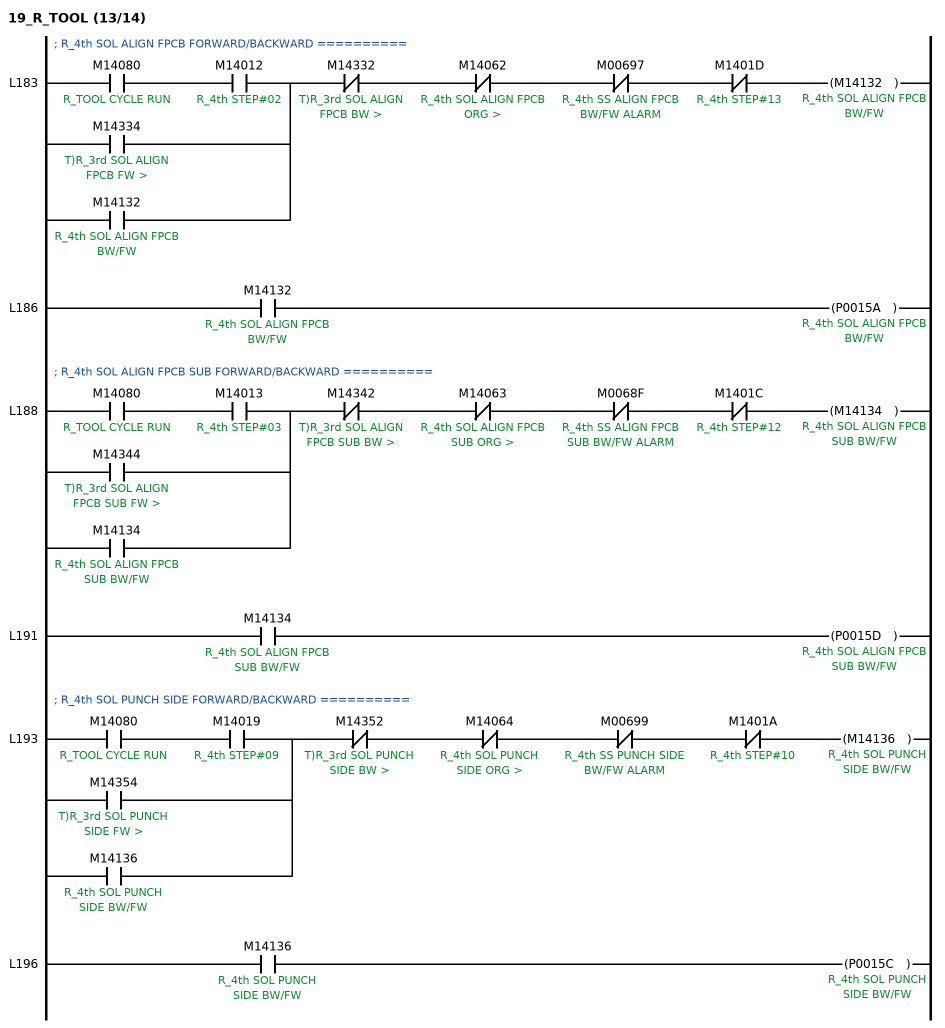
[picture p192: 19_R_TOOL rungs L183-L196]
// R_4th SOL ALIGN FPCB FORWARD/BACKWARD ==========
; L183
LOAD      M14080	// R_TOOL CYCLE RUN
AND       M14012	// R_4th STEP#02
OR        M14334	// T)R_3rd SOL ALIGN FPCB FW >
OR        M14132	// R_4th SOL ALIGN FPCB BW/FW
AND NOT   M14332	// T)R_3rd SOL ALIGN FPCB BW >
AND NOT   M14062	// R_4th SOL ALIGN FPCB ORG >
AND NOT   M00697	// R_4th SS ALIGN FPCB BW/FW ALARM
AND NOT   M1401D	// R_4th STEP#13
OUT       M14132	// R_4th SOL ALIGN FPCB BW/FW
; L186
LOAD      M14132	// R_4th SOL ALIGN FPCB BW/FW
OUT       P0015A	// R_4th SOL ALIGN FPCB BW/FW
// R_4th SOL ALIGN FPCB SUB FORWARD/BACKWARD ==========
; L188
LOAD      M14080	// R_TOOL CYCLE RUN
AND       M14013	// R_4th STEP#03
OR        M14344	// T)R_3rd SOL ALIGN FPCB SUB FW >
OR        M14134	// R_4th SOL ALIGN FPCB SUB BW/FW
AND NOT   M14342	// T)R_3rd SOL ALIGN FPCB SUB BW >
AND NOT   M14063	// R_4th SOL ALIGN FPCB SUB ORG >
AND NOT   M0068F	// R_4th SS ALIGN FPCB SUB BW/FW ALARM
AND NOT   M1401C	// R_4th STEP#12
OUT       M14134	// R_4th SOL ALIGN FPCB SUB BW/FW
; L191
LOAD      M14134	// R_4th SOL ALIGN FPCB SUB BW/FW
OUT       P0015D	// R_4th SOL ALIGN FPCB SUB BW/FW
// R_4th SOL PUNCH SIDE FORWARD/BACKWARD ==========
; L193
LOAD      M14080	// R_TOOL CYCLE RUN
AND       M14019	// R_4th STEP#09
OR        M14354	// T)R_3rd SOL PUNCH SIDE FW >
OR        M14136	// R_4th SOL PUNCH SIDE BW/FW
AND NOT   M14352	// T)R_3rd SOL PUNCH SIDE BW >
AND NOT   M14064	// R_4th SOL PUNCH SIDE ORG >
AND NOT   M00699	// R_4th SS PUNCH SIDE BW/FW ALARM
AND NOT   M1401A	// R_4th STEP#10
OUT       M14136	// R_4th SOL PUNCH SIDE BW/FW
; L196
LOAD      M14136	// R_4th SOL PUNCH SIDE BW/FW
OUT       P0015C	// R_4th SOL PUNCH SIDE BW/FW

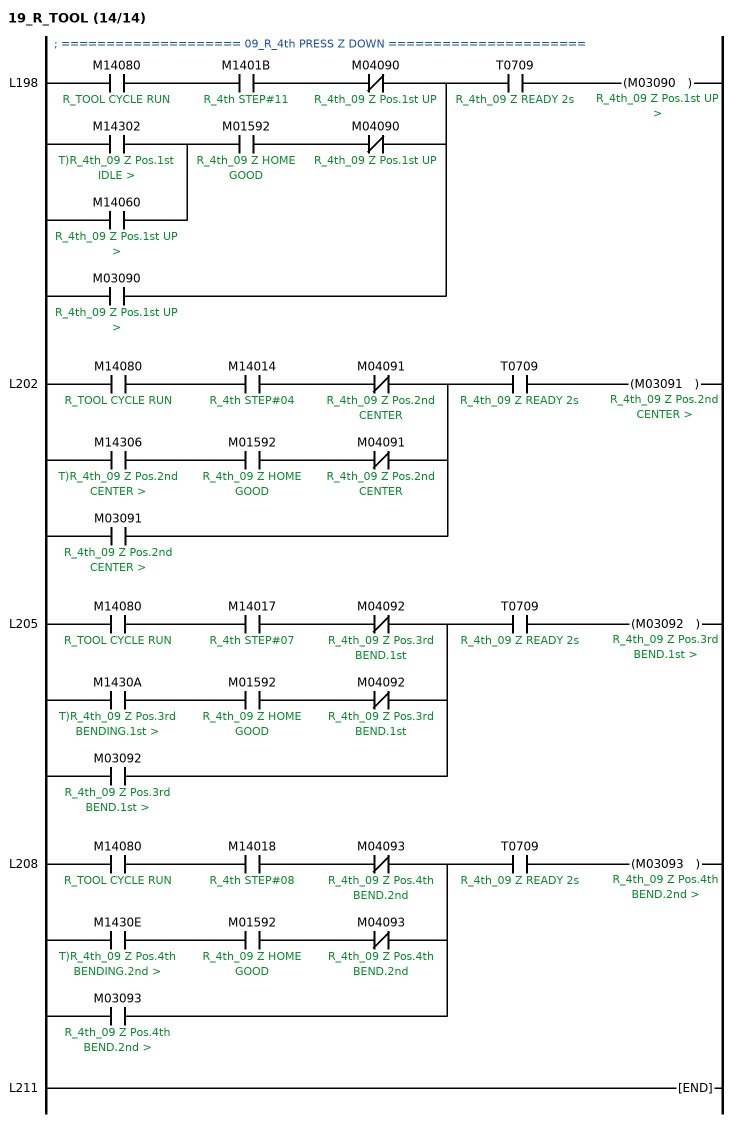
// ==================== 09_R_4th PRESS Z DOWN ======================
; L198
LOAD      M14080	// R_TOOL CYCLE RUN
AND       M1401B	// R_4th STEP#11
AND NOT   M04090	// R_4th_09 Z Pos.1st UP
LOAD      M14302	// T)R_4th_09 Z Pos.1st IDLE >
OR        M14060	// R_4th_09 Z Pos.1st UP >
AND       M01592	// R_4th_09 Z HOME GOOD
AND NOT   M04090	// R_4th_09 Z Pos.1st UP
OR LOAD
OR        M03090	// R_4th_09 Z Pos.1st UP >
AND       T0709	// R_4th_09 Z READY 2s
OUT       M03090	// R_4th_09 Z Pos.1st UP >
; L202
LOAD      M14080	// R_TOOL CYCLE RUN
AND       M14014	// R_4th STEP#04
AND NOT   M04091	// R_4th_09 Z Pos.2nd CENTER
LOAD      M14306	// T)R_4th_09 Z Pos.2nd CENTER >
AND       M01592	// R_4th_09 Z HOME GOOD
AND NOT   M04091	// R_4th_09 Z Pos.2nd CENTER
OR LOAD
OR        M03091	// R_4th_09 Z Pos.2nd CENTER >
AND       T0709	// R_4th_09 Z READY 2s
OUT       M03091	// R_4th_09 Z Pos.2nd CENTER >
; L205
LOAD      M14080	// R_TOOL CYCLE RUN
AND       M14017	// R_4th STEP#07
AND NOT   M04092	// R_4th_09 Z Pos.3rd BEND.1st
LOAD      M1430A	// T)R_4th_09 Z Pos.3rd BENDING.1st >
AND       M01592	// R_4th_09 Z HOME GOOD
AND NOT   M04092	// R_4th_09 Z Pos.3rd BEND.1st
OR LOAD
OR        M03092	// R_4th_09 Z Pos.3rd BEND.1st >
AND       T0709	// R_4th_09 Z READY 2s
OUT       M03092	// R_4th_09 Z Pos.3rd BEND.1st >
; L208
LOAD      M14080	// R_TOOL CYCLE RUN
AND       M14018	// R_4th STEP#08
AND NOT   M04093	// R_4th_09 Z Pos.4th BEND.2nd
LOAD      M1430E	// T)R_4th_09 Z Pos.4th BENDING.2nd >
AND       M01592	// R_4th_09 Z HOME GOOD
AND NOT   M04093	// R_4th_09 Z Pos.4th BEND.2nd
OR LOAD
OR        M03093	// R_4th_09 Z Pos.4th BEND.2nd >
AND       T0709	// R_4th_09 Z READY 2s
OUT       M03093	// R_4th_09 Z Pos.4th BEND.2nd >
; L211
END

PROGRAM 20_R_PP (task: ½ºÄµ ÇÁ·Î±×·¥)

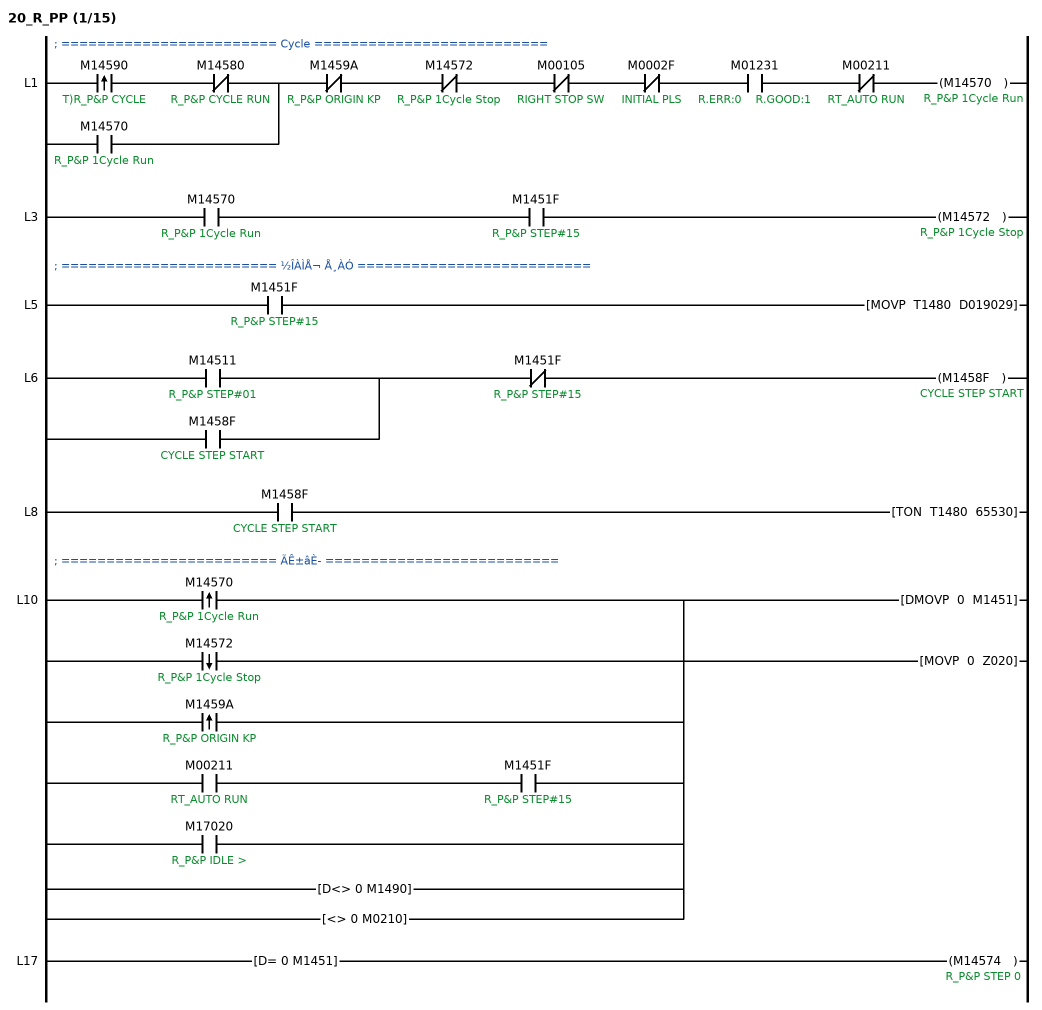
// ======================== Cycle ==========================
; L1
LOADP     M14590	// T)R_P&P CYCLE
AND NOT   M14580	// R_P&P CYCLE RUN
OR        M14570	// R_P&P 1Cycle Run
AND NOT   M1459A	// R_P&P ORIGIN KP
AND NOT   M14572	// R_P&P 1Cycle Stop
AND NOT   M00105	// RIGHT STOP SW
AND NOT   M0002F	// INITIAL PLS
AND       M01231	// R.ERR:0    R.GOOD:1
AND NOT   M00211	// RT_AUTO RUN
OUT       M14570	// R_P&P 1Cycle Run
; L3
LOAD      M14570	// R_P&P 1Cycle Run
AND       M1451F	// R_P&P STEP#15
OUT       M14572	// R_P&P 1Cycle Stop
// ======================== ½ÎÀÌÅ¬ Å¸ÀÓ ==========================
; L5
LOAD      M1451F	// R_P&P STEP#15
MOVP      T1480 D019029
; L6
LOAD      M14511	// R_P&P STEP#01
OR        M1458F	// CYCLE STEP START
AND NOT   M1451F	// R_P&P STEP#15
OUT       M1458F	// CYCLE STEP START
; L8
LOAD      M1458F	// CYCLE STEP START
TON       T1480 65530
// ======================== ÃÊ±âÈ­ ==========================
; L10
LOADP     M14570	// R_P&P 1Cycle Run
ORN       M14572	// R_P&P 1Cycle Stop
ORP       M1459A	// R_P&P ORIGIN KP
LOAD      M00211	// RT_AUTO RUN
AND       M1451F	// R_P&P STEP#15
OR LOAD
OR        M17020	// R_P&P IDLE >
ORD<>     0 M1490
OR<>      0 M0210
DMOVP     0 M1451
MOVP      0 Z020
; L17
LOADD=    0 M1451
OUT       M14574	// R_P&P STEP 0

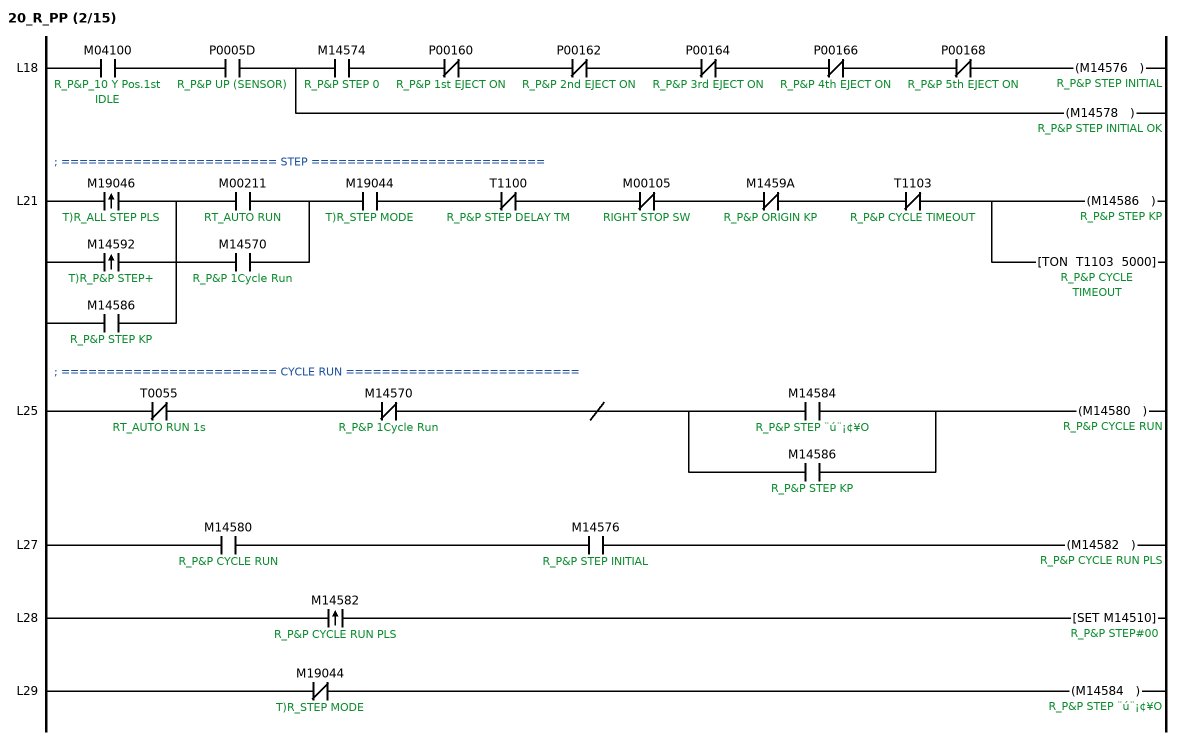
; L18
LOAD      M04100	// R_P&P_10 Y Pos.1st IDLE
AND       P0005D	// R_P&P UP (SENSOR)
MPUSH
AND       M14574	// R_P&P STEP 0
AND NOT   P00160	// R_P&P 1st EJECT ON
AND NOT   P00162	// R_P&P 2nd EJECT ON
AND NOT   P00164	// R_P&P 3rd EJECT ON
AND NOT   P00166	// R_P&P 4th EJECT ON
AND NOT   P00168	// R_P&P 5th EJECT ON
OUT       M14576	// R_P&P STEP INITIAL
MPOP
OUT       M14578	// R_P&P STEP INITIAL OK
// ======================== STEP ==========================
; L21
LOADP     M19046	// T)R_ALL STEP PLS
ORP       M14592	// T)R_P&P STEP+
OR        M14586	// R_P&P STEP KP
LOAD      M00211	// RT_AUTO RUN
OR        M14570	// R_P&P 1Cycle Run
AND LOAD
AND       M19044	// T)R_STEP MODE
AND NOT   T1100	// R_P&P STEP DELAY TM
AND NOT   M00105	// RIGHT STOP SW
AND NOT   M1459A	// R_P&P ORIGIN KP
AND NOT   T1103	// R_P&P CYCLE TIMEOUT
OUT       M14586	// R_P&P STEP KP
TON       T1103 5000	// R_P&P CYCLE TIMEOUT
// ======================== CYCLE RUN ==========================
; L25
LOAD NOT  T0055	// RT_AUTO RUN 1s
AND NOT   M14570	// R_P&P 1Cycle Run
NOT
LOAD      M14584	// R_P&P STEP ¨ú¨¡¢¥O
OR        M14586	// R_P&P STEP KP
AND LOAD
OUT       M14580	// R_P&P CYCLE RUN
; L27
LOAD      M14580	// R_P&P CYCLE RUN
AND       M14576	// R_P&P STEP INITIAL
OUT       M14582	// R_P&P CYCLE RUN PLS
; L28
LOADP     M14582	// R_P&P CYCLE RUN PLS
SET       M14510	// R_P&P STEP#00
; L29
LOAD NOT  M19044	// T)R_STEP MODE
OUT       M14584	// R_P&P STEP ¨ú¨¡¢¥O

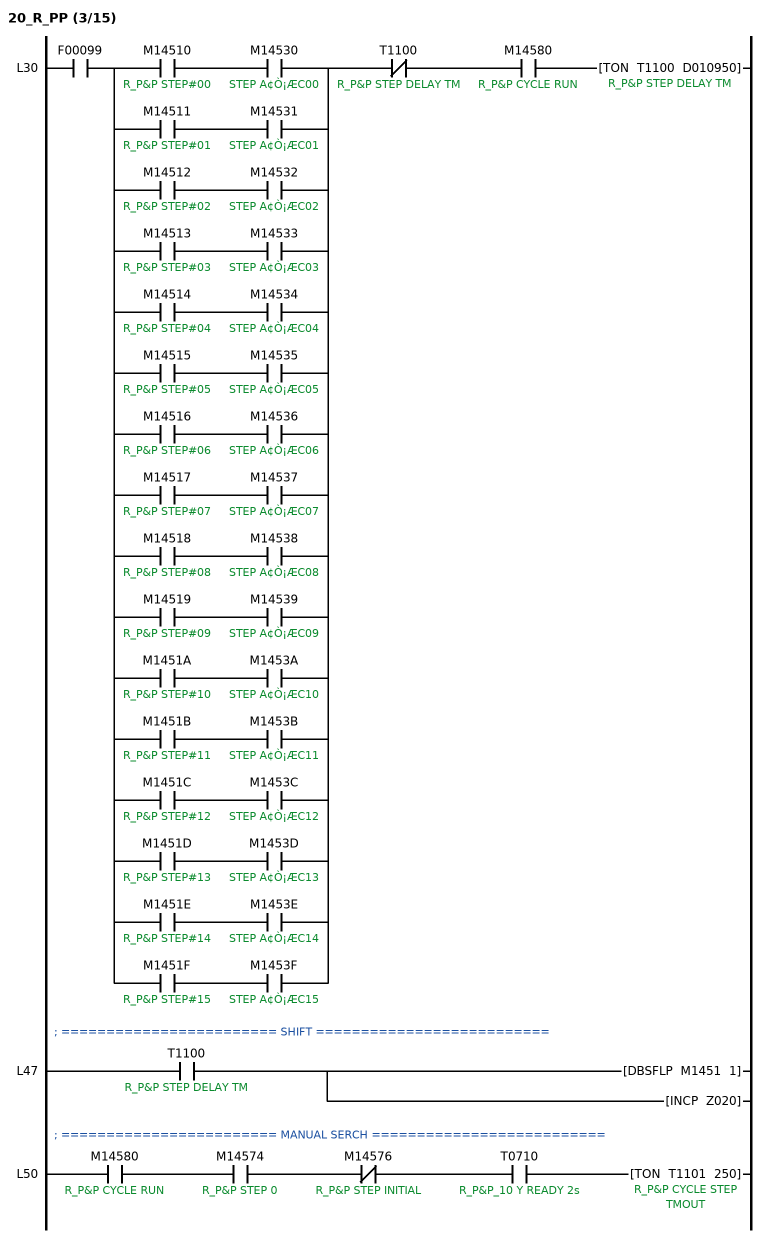
; L30
LOAD      F00099
LOAD      M14510	// R_P&P STEP#00
AND       M14530	// STEP A¢Ò¡ÆC00
LOAD      M14511	// R_P&P STEP#01
AND       M14531	// STEP A¢Ò¡ÆC01
OR LOAD
LOAD      M14512	// R_P&P STEP#02
AND       M14532	// STEP A¢Ò¡ÆC02
OR LOAD
LOAD      M14513	// R_P&P STEP#03
AND       M14533	// STEP A¢Ò¡ÆC03
OR LOAD
LOAD      M14514	// R_P&P STEP#04
AND       M14534	// STEP A¢Ò¡ÆC04
OR LOAD
LOAD      M14515	// R_P&P STEP#05
AND       M14535	// STEP A¢Ò¡ÆC05
OR LOAD
LOAD      M14516	// R_P&P STEP#06
AND       M14536	// STEP A¢Ò¡ÆC06
OR LOAD
LOAD      M14517	// R_P&P STEP#07
AND       M14537	// STEP A¢Ò¡ÆC07
OR LOAD
LOAD      M14518	// R_P&P STEP#08
AND       M14538	// STEP A¢Ò¡ÆC08
OR LOAD
LOAD      M14519	// R_P&P STEP#09
AND       M14539	// STEP A¢Ò¡ÆC09
OR LOAD
LOAD      M1451A	// R_P&P STEP#10
AND       M1453A	// STEP A¢Ò¡ÆC10
OR LOAD
LOAD      M1451B	// R_P&P STEP#11
AND       M1453B	// STEP A¢Ò¡ÆC11
OR LOAD
LOAD      M1451C	// R_P&P STEP#12
AND       M1453C	// STEP A¢Ò¡ÆC12
OR LOAD
LOAD      M1451D	// R_P&P STEP#13
AND       M1453D	// STEP A¢Ò¡ÆC13
OR LOAD
LOAD      M1451E	// R_P&P STEP#14
AND       M1453E	// STEP A¢Ò¡ÆC14
OR LOAD
LOAD      M1451F	// R_P&P STEP#15
AND       M1453F	// STEP A¢Ò¡ÆC15
OR LOAD
AND LOAD
AND NOT   T1100	// R_P&P STEP DELAY TM
AND       M14580	// R_P&P CYCLE RUN
TON       T1100 D010950	// R_P&P STEP DELAY TM
// ======================== SHIFT ==========================
; L47
LOAD      T1100	// R_P&P STEP DELAY TM
DBSFLP    M1451 1
INCP      Z020
// ======================== MANUAL SERCH ==========================
; L50
LOAD      M14580	// R_P&P CYCLE RUN
AND       M14574	// R_P&P STEP 0
AND NOT   M14576	// R_P&P STEP INITIAL
AND       T0710	// R_P&P_10 Y READY 2s
TON       T1101 250	// R_P&P CYCLE STEP TMOUT

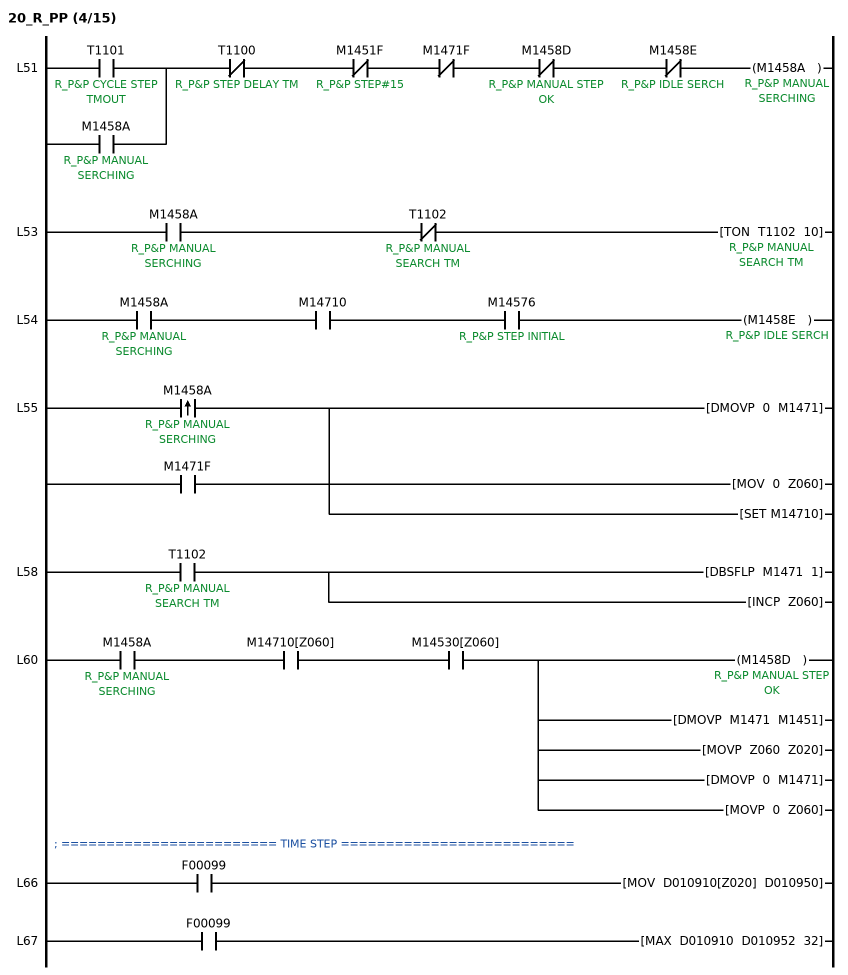
; L51
LOAD      T1101	// R_P&P CYCLE STEP TMOUT
OR        M1458A	// R_P&P MANUAL SERCHING
AND NOT   T1100	// R_P&P STEP DELAY TM
AND NOT   M1451F	// R_P&P STEP#15
AND NOT   M1471F
AND NOT   M1458D	// R_P&P MANUAL STEP OK
AND NOT   M1458E	// R_P&P IDLE SERCH
OUT       M1458A	// R_P&P MANUAL SERCHING
; L53
LOAD      M1458A	// R_P&P MANUAL SERCHING
AND NOT   T1102	// R_P&P MANUAL SEARCH TM
TON       T1102 10	// R_P&P MANUAL SEARCH TM
; L54
LOAD      M1458A	// R_P&P MANUAL SERCHING
AND       M14710
AND       M14576	// R_P&P STEP INITIAL
OUT       M1458E	// R_P&P IDLE SERCH
; L55
LOADP     M1458A	// R_P&P MANUAL SERCHING
OR        M1471F
DMOVP     0 M1471
MOV       0 Z060
SET       M14710
; L58
LOAD      T1102	// R_P&P MANUAL SEARCH TM
DBSFLP    M1471 1
INCP      Z060
; L60
LOAD      M1458A	// R_P&P MANUAL SERCHING
AND       M14710[Z060]
AND       M14530[Z060]
OUT       M1458D	// R_P&P MANUAL STEP OK
DMOVP     M1471 M1451
MOVP      Z060 Z020
DMOVP     0 M1471
MOVP      0 Z060
// ======================== TIME STEP ==========================
; L66
LOAD      F00099
MOV       D010910[Z020] D010950
; L67
LOAD      F00099
MAX       D010910 D010952 32

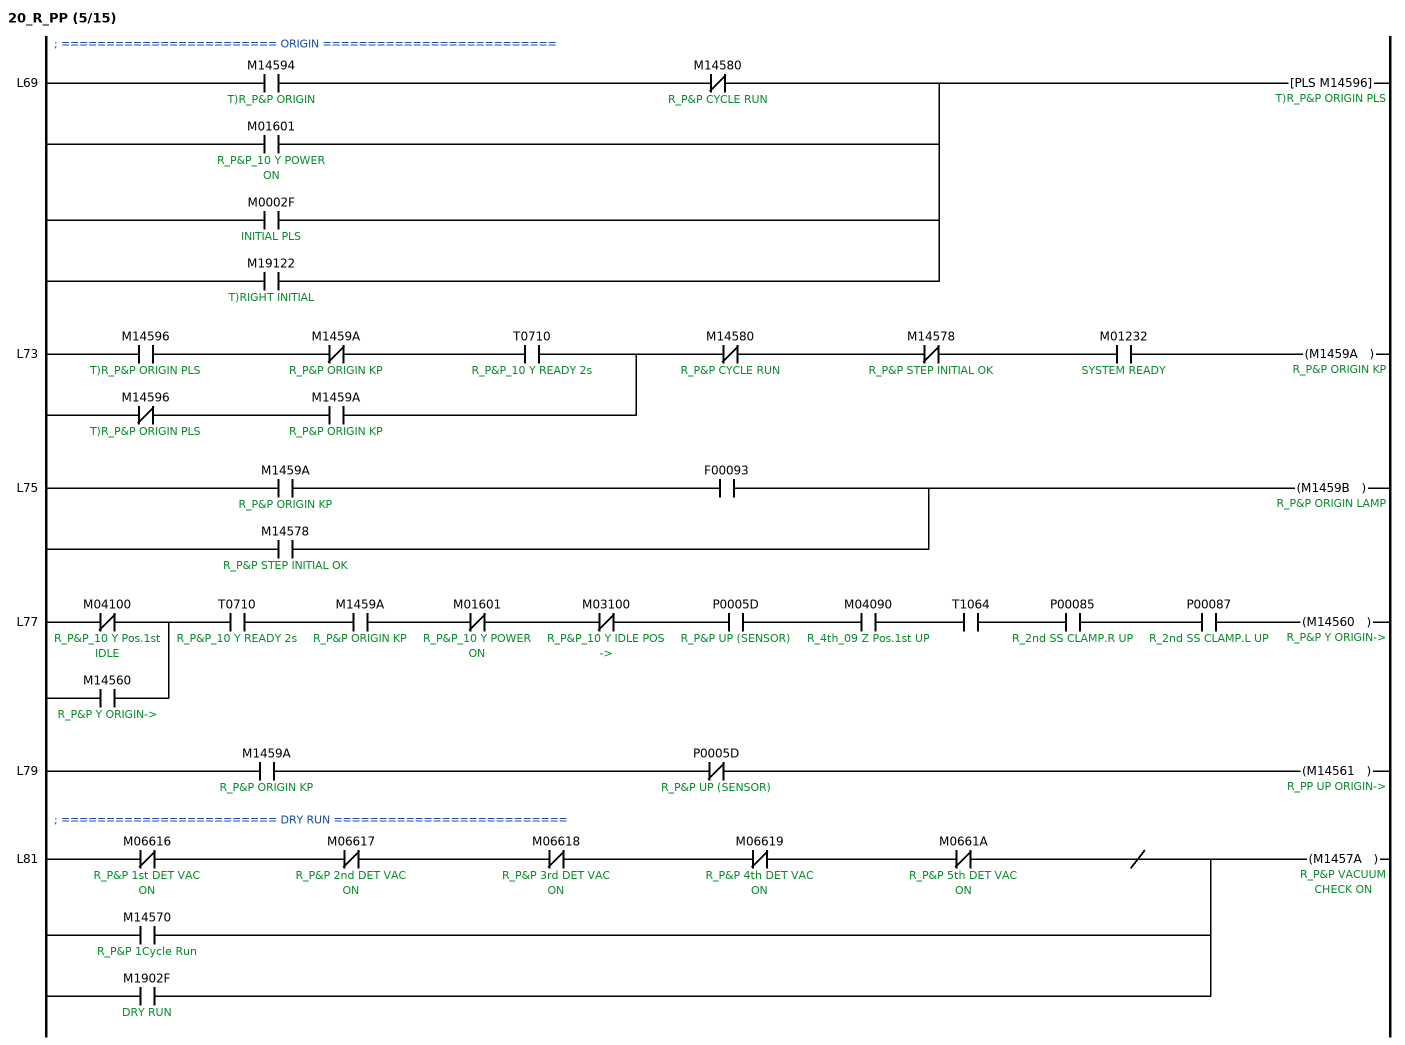
// ======================== ORIGIN ==========================
; L69
LOAD      M14594	// T)R_P&P ORIGIN
AND NOT   M14580	// R_P&P CYCLE RUN
OR        M01601	// R_P&P_10 Y POWER ON
OR        M0002F	// INITIAL PLS
OR        M19122	// T)RIGHT INITIAL
OUTP      M14596	// T)R_P&P ORIGIN PLS
; L73
LOAD      M14596	// T)R_P&P ORIGIN PLS
AND NOT   M1459A	// R_P&P ORIGIN KP
AND       T0710	// R_P&P_10 Y READY 2s
LOAD NOT  M14596	// T)R_P&P ORIGIN PLS
AND       M1459A	// R_P&P ORIGIN KP
OR LOAD
AND NOT   M14580	// R_P&P CYCLE RUN
AND NOT   M14578	// R_P&P STEP INITIAL OK
AND       M01232	// SYSTEM READY
OUT       M1459A	// R_P&P ORIGIN KP
; L75
LOAD      M1459A	// R_P&P ORIGIN KP
AND       F00093
OR        M14578	// R_P&P STEP INITIAL OK
OUT       M1459B	// R_P&P ORIGIN LAMP
; L77
LOAD NOT  M04100	// R_P&P_10 Y Pos.1st IDLE
OR        M14560	// R_P&P Y ORIGIN->
AND       T0710	// R_P&P_10 Y READY 2s
AND       M1459A	// R_P&P ORIGIN KP
AND NOT   M01601	// R_P&P_10 Y POWER ON
AND NOT   M03100	// R_P&P_10 Y IDLE POS ->
AND       P0005D	// R_P&P UP (SENSOR)
AND       M04090	// R_4th_09 Z Pos.1st UP
AND       T1064
AND       P00085	// R_2nd SS CLAMP.R UP
AND       P00087	// R_2nd SS CLAMP.L UP
OUT       M14560	// R_P&P Y ORIGIN->
; L79
LOAD      M1459A	// R_P&P ORIGIN KP
AND NOT   P0005D	// R_P&P UP (SENSOR)
OUT       M14561	// R_PP UP ORIGIN->
// ======================== DRY RUN ==========================
; L81
LOAD NOT  M06616	// R_P&P 1st DET VAC ON
AND NOT   M06617	// R_P&P 2nd DET VAC ON
AND NOT   M06618	// R_P&P 3rd DET VAC ON
AND NOT   M06619	// R_P&P 4th DET VAC ON
AND NOT   M0661A	// R_P&P 5th DET VAC ON
NOT
OR        M14570	// R_P&P 1Cycle Run
OR        M1902F	// DRY RUN
OUT       M1457A	// R_P&P VACUUM CHECK ON

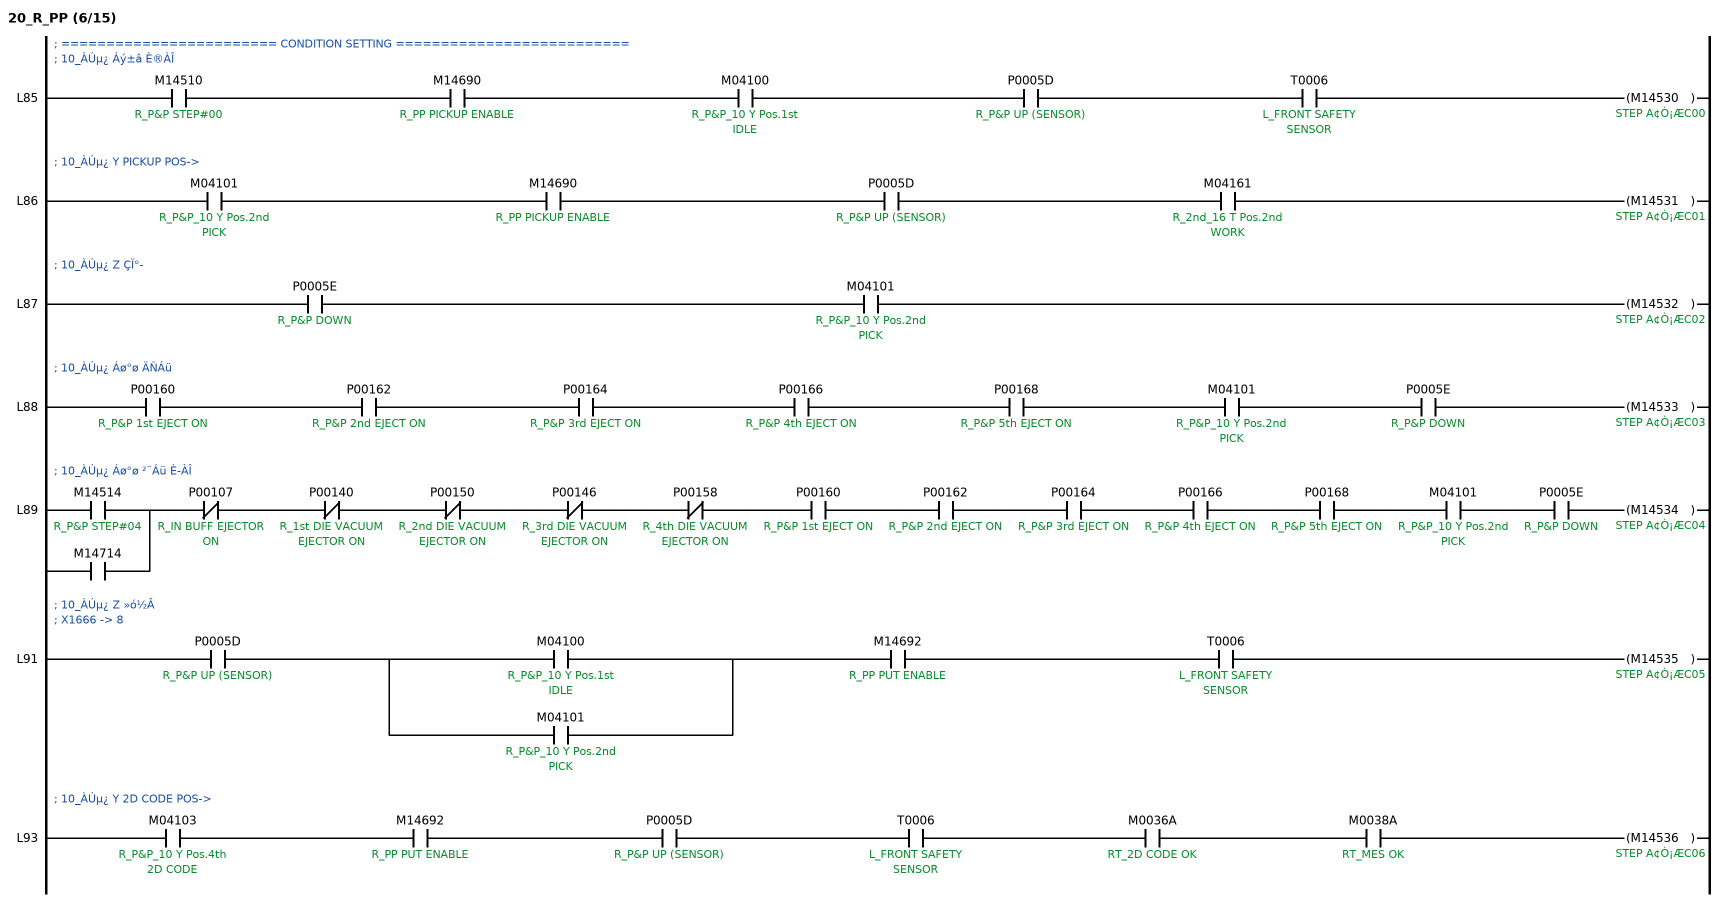
// ======================== CONDITION SETTING ==========================
; L85
LOAD      M14510	// R_P&P STEP#00
AND       M14690	// R_PP PICKUP ENABLE
AND       M04100	// R_P&P_10 Y Pos.1st IDLE
AND       P0005D	// R_P&P UP (SENSOR)
AND       T0006	// L_FRONT SAFETY SENSOR
OUT       M14530	// STEP A¢Ò¡ÆC00
// output comment: 10_ÀÚµ¿ Áý±â È®ÀÎ
; L86
LOAD      M04101	// R_P&P_10 Y Pos.2nd PICK
AND       M14690	// R_PP PICKUP ENABLE
AND       P0005D	// R_P&P UP (SENSOR)
AND       M04161	// R_2nd_16 T Pos.2nd WORK
OUT       M14531	// STEP A¢Ò¡ÆC01
// output comment: 10_ÀÚµ¿ Y PICKUP POS->
; L87
LOAD      P0005E	// R_P&P DOWN
AND       M04101	// R_P&P_10 Y Pos.2nd PICK
OUT       M14532	// STEP A¢Ò¡ÆC02
// output comment: 10_ÀÚµ¿ Z ÇÏ°­
; L88
LOAD      P00160	// R_P&P 1st EJECT ON
AND       P00162	// R_P&P 2nd EJECT ON
AND       P00164	// R_P&P 3rd EJECT ON
AND       P00166	// R_P&P 4th EJECT ON
AND       P00168	// R_P&P 5th EJECT ON
AND       M04101	// R_P&P_10 Y Pos.2nd PICK
AND       P0005E	// R_P&P DOWN
OUT       M14533	// STEP A¢Ò¡ÆC03
// output comment: 10_ÀÚµ¿ Áø°ø ÄÑÁü
; L89
LOAD      M14514	// R_P&P STEP#04
OR        M14714
AND NOT   P00107	// R_IN BUFF EJECTOR ON
AND NOT   P00140	// R_1st DIE VACUUM EJECTOR ON
AND NOT   P00150	// R_2nd DIE VACUUM EJECTOR ON
AND NOT   P00146	// R_3rd DIE VACUUM EJECTOR ON
AND NOT   P00158	// R_4th DIE VACUUM EJECTOR ON
AND       P00160	// R_P&P 1st EJECT ON
AND       P00162	// R_P&P 2nd EJECT ON
AND       P00164	// R_P&P 3rd EJECT ON
AND       P00166	// R_P&P 4th EJECT ON
AND       P00168	// R_P&P 5th EJECT ON
AND       M04101	// R_P&P_10 Y Pos.2nd PICK
AND       P0005E	// R_P&P DOWN
OUT       M14534	// STEP A¢Ò¡ÆC04
// output comment: 10_ÀÚµ¿ Áø°ø ²¨Áü È­ÀÎ
; L91
LOAD      P0005D	// R_P&P UP (SENSOR)
LOAD      M04100	// R_P&P_10 Y Pos.1st IDLE
OR        M04101	// R_P&P_10 Y Pos.2nd PICK
AND LOAD
AND       M14692	// R_PP PUT ENABLE
AND       T0006	// L_FRONT SAFETY SENSOR
OUT       M14535	// STEP A¢Ò¡ÆC05
// output comment: 10_ÀÚµ¿ Z »ó½Â X1666 -> 8
; L93
LOAD      M04103	// R_P&P_10 Y Pos.4th 2D CODE
AND       M14692	// R_PP PUT ENABLE
AND       P0005D	// R_P&P UP (SENSOR)
AND       T0006	// L_FRONT SAFETY SENSOR
AND       M0036A	// RT_2D CODE OK
AND       M0038A	// RT_MES OK
OUT       M14536	// STEP A¢Ò¡ÆC06
// output comment: 10_ÀÚµ¿ Y 2D CODE POS->

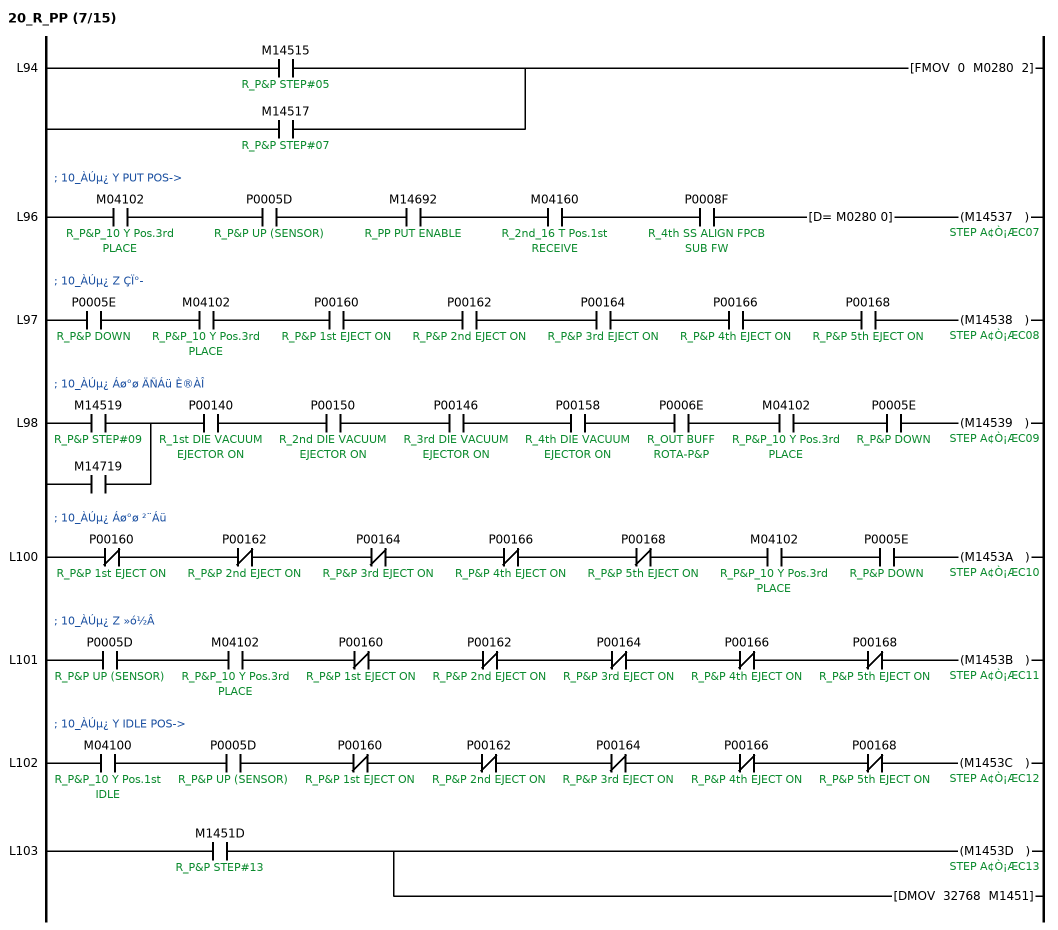
; L94
LOAD      M14515	// R_P&P STEP#05
OR        M14517	// R_P&P STEP#07
FMOV      0 M0280 2
; L96
LOAD      M04102	// R_P&P_10 Y Pos.3rd PLACE
AND       P0005D	// R_P&P UP (SENSOR)
AND       M14692	// R_PP PUT ENABLE
AND       M04160	// R_2nd_16 T Pos.1st RECEIVE
AND       P0008F	// R_4th SS ALIGN FPCB SUB FW
ANDD=     M0280 0
OUT       M14537	// STEP A¢Ò¡ÆC07
// output comment: 10_ÀÚµ¿ Y PUT POS->
; L97
LOAD      P0005E	// R_P&P DOWN
AND       M04102	// R_P&P_10 Y Pos.3rd PLACE
AND       P00160	// R_P&P 1st EJECT ON
AND       P00162	// R_P&P 2nd EJECT ON
AND       P00164	// R_P&P 3rd EJECT ON
AND       P00166	// R_P&P 4th EJECT ON
AND       P00168	// R_P&P 5th EJECT ON
OUT       M14538	// STEP A¢Ò¡ÆC08
// output comment: 10_ÀÚµ¿ Z ÇÏ°­
; L98
LOAD      M14519	// R_P&P STEP#09
OR        M14719
AND       P00140	// R_1st DIE VACUUM EJECTOR ON
AND       P00150	// R_2nd DIE VACUUM EJECTOR ON
AND       P00146	// R_3rd DIE VACUUM EJECTOR ON
AND       P00158	// R_4th DIE VACUUM EJECTOR ON
AND       P0006E	// R_OUT BUFF ROTA-P&P
AND       M04102	// R_P&P_10 Y Pos.3rd PLACE
AND       P0005E	// R_P&P DOWN
OUT       M14539	// STEP A¢Ò¡ÆC09
// output comment: 10_ÀÚµ¿ Áø°ø ÄÑÁü È®ÀÎ
; L100
LOAD NOT  P00160	// R_P&P 1st EJECT ON
AND NOT   P00162	// R_P&P 2nd EJECT ON
AND NOT   P00164	// R_P&P 3rd EJECT ON
AND NOT   P00166	// R_P&P 4th EJECT ON
AND NOT   P00168	// R_P&P 5th EJECT ON
AND       M04102	// R_P&P_10 Y Pos.3rd PLACE
AND       P0005E	// R_P&P DOWN
OUT       M1453A	// STEP A¢Ò¡ÆC10
// output comment: 10_ÀÚµ¿ Áø°ø ²¨Áü
; L101
LOAD      P0005D	// R_P&P UP (SENSOR)
AND       M04102	// R_P&P_10 Y Pos.3rd PLACE
AND NOT   P00160	// R_P&P 1st EJECT ON
AND NOT   P00162	// R_P&P 2nd EJECT ON
AND NOT   P00164	// R_P&P 3rd EJECT ON
AND NOT   P00166	// R_P&P 4th EJECT ON
AND NOT   P00168	// R_P&P 5th EJECT ON
OUT       M1453B	// STEP A¢Ò¡ÆC11
// output comment: 10_ÀÚµ¿ Z »ó½Â
; L102
LOAD      M04100	// R_P&P_10 Y Pos.1st IDLE
AND       P0005D	// R_P&P UP (SENSOR)
AND NOT   P00160	// R_P&P 1st EJECT ON
AND NOT   P00162	// R_P&P 2nd EJECT ON
AND NOT   P00164	// R_P&P 3rd EJECT ON
AND NOT   P00166	// R_P&P 4th EJECT ON
AND NOT   P00168	// R_P&P 5th EJECT ON
OUT       M1453C	// STEP A¢Ò¡ÆC12
// output comment: 10_ÀÚµ¿ Y IDLE POS->
; L103
LOAD      M1451D	// R_P&P STEP#13
OUT       M1453D	// STEP A¢Ò¡ÆC13
DMOV      32768 M1451

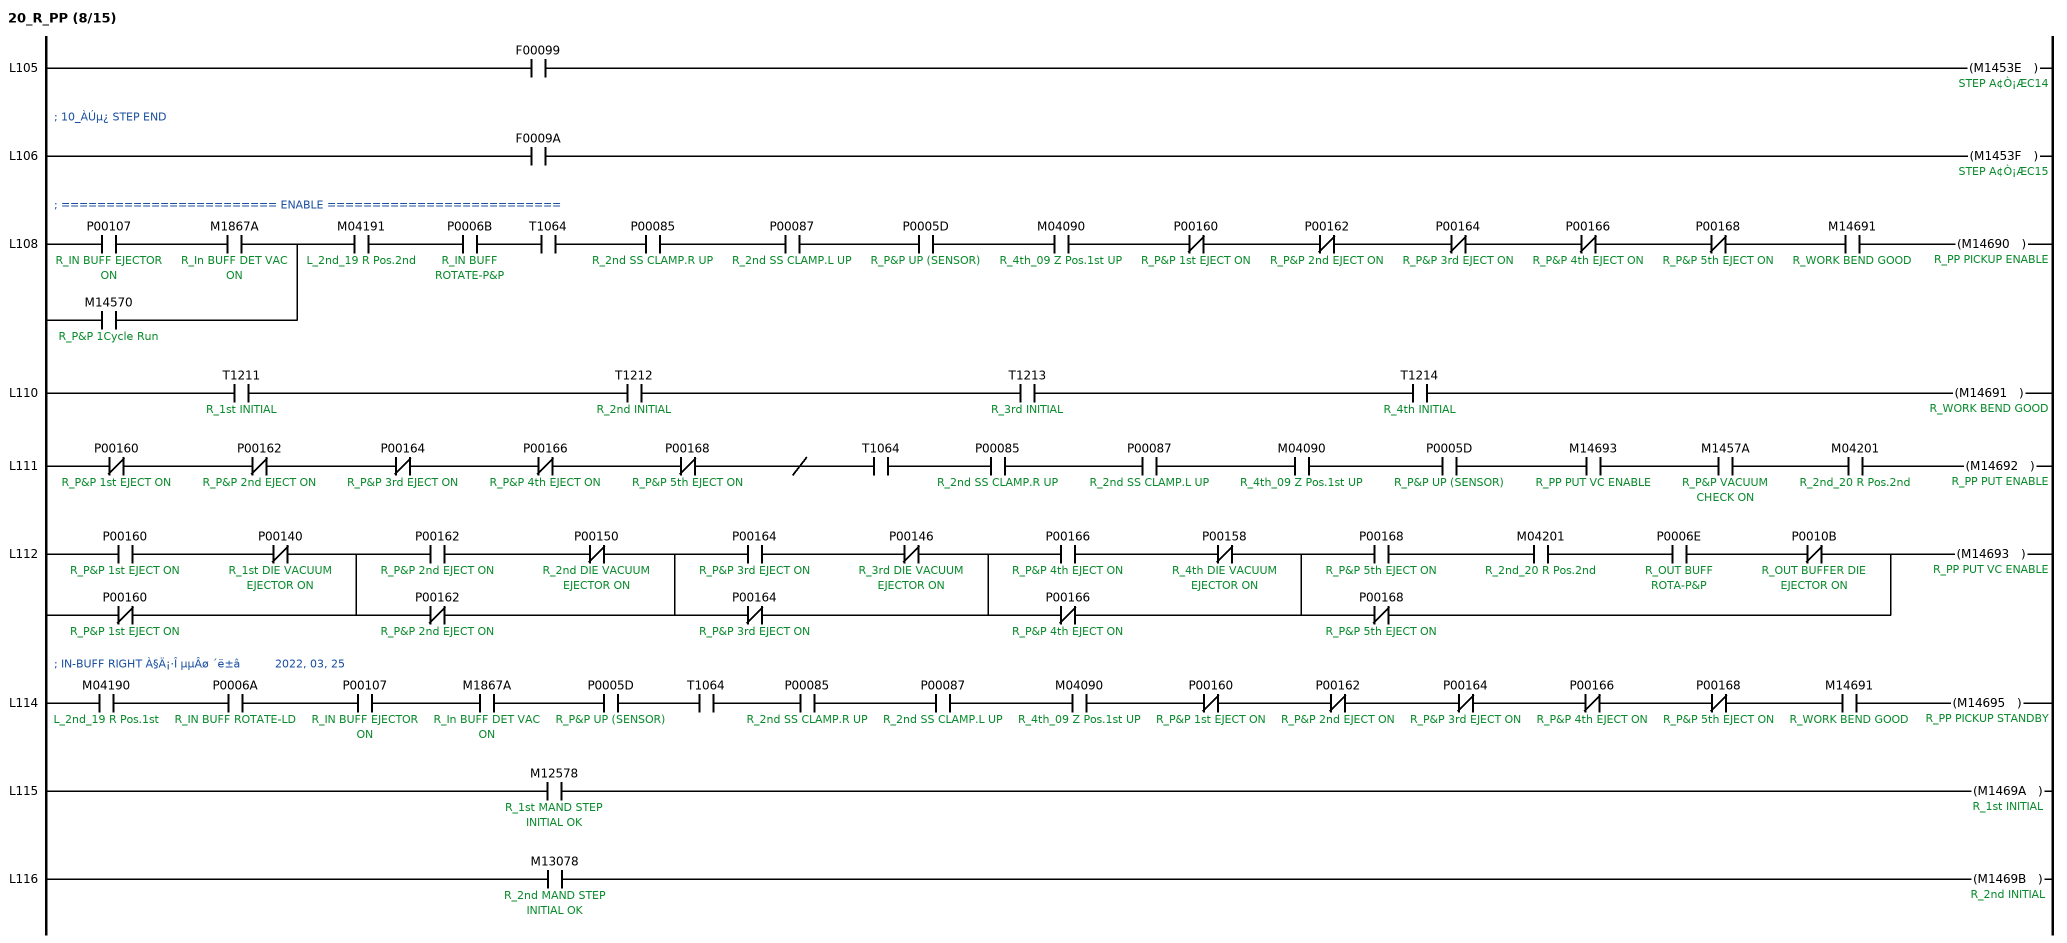
; L105
LOAD      F00099
OUT       M1453E	// STEP A¢Ò¡ÆC14
; L106
LOAD      F0009A
OUT       M1453F	// STEP A¢Ò¡ÆC15
// output comment: 10_ÀÚµ¿ STEP END
// ======================== ENABLE ==========================
; L108
LOAD      P00107	// R_IN BUFF EJECTOR ON
AND       M1867A	// R_In BUFF DET VAC ON
OR        M14570	// R_P&P 1Cycle Run
AND       M04191	// L_2nd_19 R Pos.2nd
AND       P0006B	// R_IN BUFF ROTATE-P&P
AND       T1064
AND       P00085	// R_2nd SS CLAMP.R UP
AND       P00087	// R_2nd SS CLAMP.L UP
AND       P0005D	// R_P&P UP (SENSOR)
AND       M04090	// R_4th_09 Z Pos.1st UP
AND NOT   P00160	// R_P&P 1st EJECT ON
AND NOT   P00162	// R_P&P 2nd EJECT ON
AND NOT   P00164	// R_P&P 3rd EJECT ON
AND NOT   P00166	// R_P&P 4th EJECT ON
AND NOT   P00168	// R_P&P 5th EJECT ON
AND       M14691	// R_WORK BEND GOOD
OUT       M14690	// R_PP PICKUP ENABLE
; L110
LOAD      T1211	// R_1st INITIAL
AND       T1212	// R_2nd INITIAL
AND       T1213	// R_3rd INITIAL
AND       T1214	// R_4th INITIAL
OUT       M14691	// R_WORK BEND GOOD
; L111
LOAD NOT  P00160	// R_P&P 1st EJECT ON
AND NOT   P00162	// R_P&P 2nd EJECT ON
AND NOT   P00164	// R_P&P 3rd EJECT ON
AND NOT   P00166	// R_P&P 4th EJECT ON
AND NOT   P00168	// R_P&P 5th EJECT ON
NOT
AND       T1064
AND       P00085	// R_2nd SS CLAMP.R UP
AND       P00087	// R_2nd SS CLAMP.L UP
AND       M04090	// R_4th_09 Z Pos.1st UP
AND       P0005D	// R_P&P UP (SENSOR)
AND       M14693	// R_PP PUT VC ENABLE
AND       M1457A	// R_P&P VACUUM CHECK ON
AND       M04201	// R_2nd_20 R Pos.2nd
OUT       M14692	// R_PP PUT ENABLE
; L112
LOAD      P00160	// R_P&P 1st EJECT ON
AND NOT   P00140	// R_1st DIE VACUUM EJECTOR ON
OR NOT    P00160	// R_P&P 1st EJECT ON
LOAD      P00162	// R_P&P 2nd EJECT ON
AND NOT   P00150	// R_2nd DIE VACUUM EJECTOR ON
OR NOT    P00162	// R_P&P 2nd EJECT ON
AND LOAD
LOAD      P00164	// R_P&P 3rd EJECT ON
AND NOT   P00146	// R_3rd DIE VACUUM EJECTOR ON
OR NOT    P00164	// R_P&P 3rd EJECT ON
AND LOAD
LOAD      P00166	// R_P&P 4th EJECT ON
AND NOT   P00158	// R_4th DIE VACUUM EJECTOR ON
OR NOT    P00166	// R_P&P 4th EJECT ON
AND LOAD
LOAD      P00168	// R_P&P 5th EJECT ON
AND       M04201	// R_2nd_20 R Pos.2nd
AND       P0006E	// R_OUT BUFF ROTA-P&P
AND NOT   P0010B	// R_OUT BUFFER DIE EJECTOR ON
OR NOT    P00168	// R_P&P 5th EJECT ON
AND LOAD
OUT       M14693	// R_PP PUT VC ENABLE
; L114
LOAD      M04190	// L_2nd_19 R Pos.1st 
AND       P0006A	// R_IN BUFF ROTATE-LD
AND       P00107	// R_IN BUFF EJECTOR ON
AND       M1867A	// R_In BUFF DET VAC ON
AND       P0005D	// R_P&P UP (SENSOR)
AND       T1064
AND       P00085	// R_2nd SS CLAMP.R UP
AND       P00087	// R_2nd SS CLAMP.L UP
AND       M04090	// R_4th_09 Z Pos.1st UP
AND NOT   P00160	// R_P&P 1st EJECT ON
AND NOT   P00162	// R_P&P 2nd EJECT ON
AND NOT   P00164	// R_P&P 3rd EJECT ON
AND NOT   P00166	// R_P&P 4th EJECT ON
AND NOT   P00168	// R_P&P 5th EJECT ON
AND       M14691	// R_WORK BEND GOOD
OUT       M14695	// R_PP PICKUP STANDBY
// output comment: IN-BUFF RIGHT À§Ä¡·Î µµÂø ´ë±â          2022, 03, 25
; L115
LOAD      M12578	// R_1st MAND STEP INITIAL OK
OUT       M1469A	// R_1st INITIAL
; L116
LOAD      M13078	// R_2nd MAND STEP INITIAL OK
OUT       M1469B	// R_2nd INITIAL

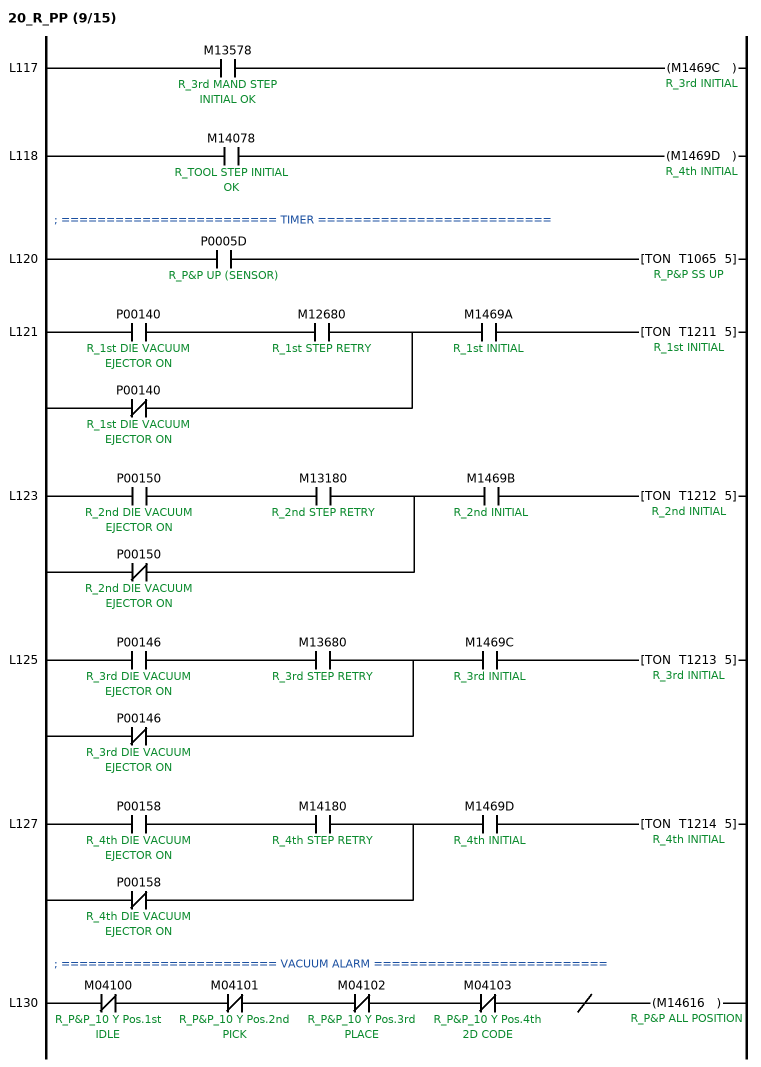
; L117
LOAD      M13578	// R_3rd MAND STEP INITIAL OK
OUT       M1469C	// R_3rd INITIAL
; L118
LOAD      M14078	// R_TOOL STEP INITIAL OK
OUT       M1469D	// R_4th INITIAL
// ======================== TIMER ==========================
; L120
LOAD      P0005D	// R_P&P UP (SENSOR)
TON       T1065 5	// R_P&P SS UP
; L121
LOAD      P00140	// R_1st DIE VACUUM EJECTOR ON
AND       M12680	// R_1st STEP RETRY
OR NOT    P00140	// R_1st DIE VACUUM EJECTOR ON
AND       M1469A	// R_1st INITIAL
TON       T1211 5	// R_1st INITIAL
; L123
LOAD      P00150	// R_2nd DIE VACUUM EJECTOR ON
AND       M13180	// R_2nd STEP RETRY
OR NOT    P00150	// R_2nd DIE VACUUM EJECTOR ON
AND       M1469B	// R_2nd INITIAL
TON       T1212 5	// R_2nd INITIAL
; L125
LOAD      P00146	// R_3rd DIE VACUUM EJECTOR ON
AND       M13680	// R_3rd STEP RETRY
OR NOT    P00146	// R_3rd DIE VACUUM EJECTOR ON
AND       M1469C	// R_3rd INITIAL
TON       T1213 5	// R_3rd INITIAL
; L127
LOAD      P00158	// R_4th DIE VACUUM EJECTOR ON
AND       M14180	// R_4th STEP RETRY
OR NOT    P00158	// R_4th DIE VACUUM EJECTOR ON
AND       M1469D	// R_4th INITIAL
TON       T1214 5	// R_4th INITIAL
// ======================== VACUUM ALARM ==========================
; L130
LOAD NOT  M04100	// R_P&P_10 Y Pos.1st IDLE
AND NOT   M04101	// R_P&P_10 Y Pos.2nd PICK
AND NOT   M04102	// R_P&P_10 Y Pos.3rd PLACE
AND NOT   M04103	// R_P&P_10 Y Pos.4th 2D CODE
NOT
OUT       M14616	// R_P&P ALL POSITION

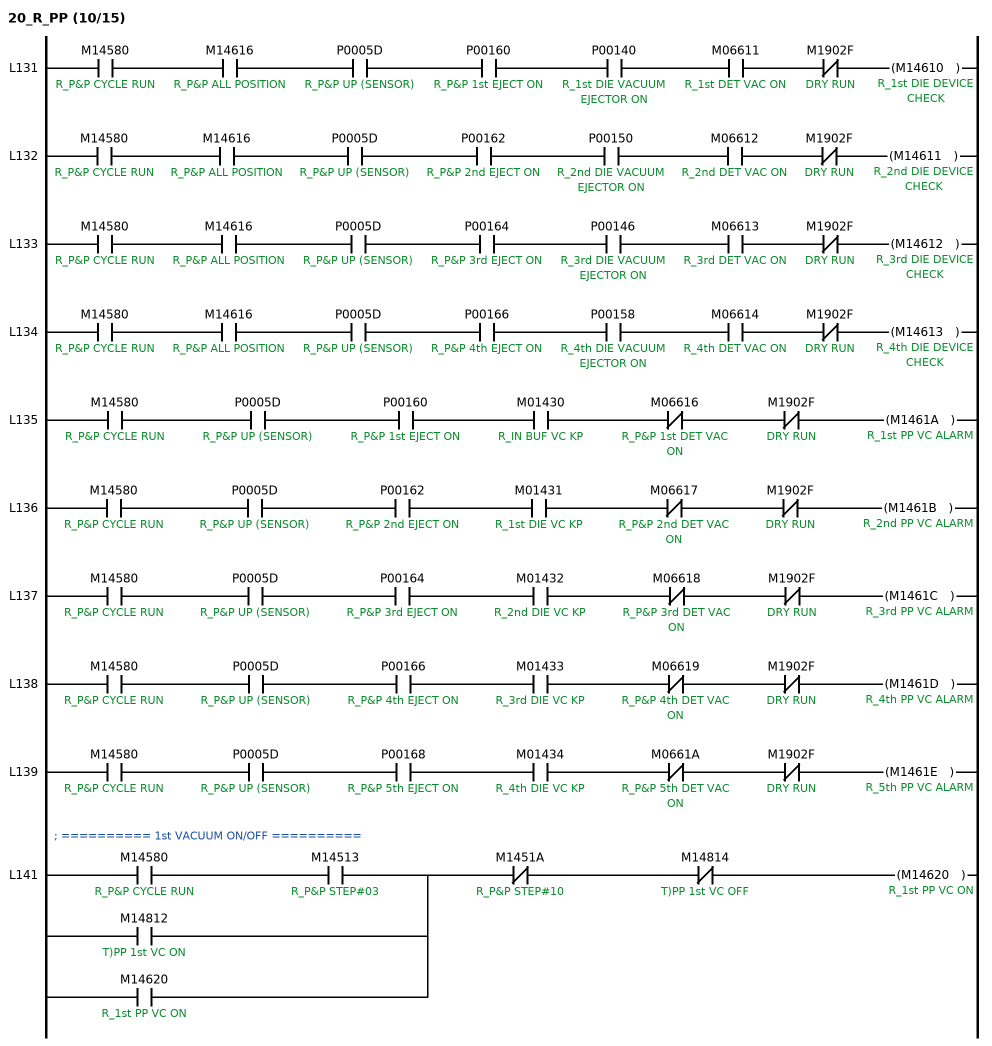
; L131
LOAD      M14580	// R_P&P CYCLE RUN
AND       M14616	// R_P&P ALL POSITION
AND       P0005D	// R_P&P UP (SENSOR)
AND       P00160	// R_P&P 1st EJECT ON
AND       P00140	// R_1st DIE VACUUM EJECTOR ON
AND       M06611	// R_1st DET VAC ON
AND NOT   M1902F	// DRY RUN
OUT       M14610	// R_1st DIE DEVICE CHECK
; L132
LOAD      M14580	// R_P&P CYCLE RUN
AND       M14616	// R_P&P ALL POSITION
AND       P0005D	// R_P&P UP (SENSOR)
AND       P00162	// R_P&P 2nd EJECT ON
AND       P00150	// R_2nd DIE VACUUM EJECTOR ON
AND       M06612	// R_2nd DET VAC ON
AND NOT   M1902F	// DRY RUN
OUT       M14611	// R_2nd DIE DEVICE CHECK
; L133
LOAD      M14580	// R_P&P CYCLE RUN
AND       M14616	// R_P&P ALL POSITION
AND       P0005D	// R_P&P UP (SENSOR)
AND       P00164	// R_P&P 3rd EJECT ON
AND       P00146	// R_3rd DIE VACUUM EJECTOR ON
AND       M06613	// R_3rd DET VAC ON
AND NOT   M1902F	// DRY RUN
OUT       M14612	// R_3rd DIE DEVICE CHECK
; L134
LOAD      M14580	// R_P&P CYCLE RUN
AND       M14616	// R_P&P ALL POSITION
AND       P0005D	// R_P&P UP (SENSOR)
AND       P00166	// R_P&P 4th EJECT ON
AND       P00158	// R_4th DIE VACUUM EJECTOR ON
AND       M06614	// R_4th DET VAC ON
AND NOT   M1902F	// DRY RUN
OUT       M14613	// R_4th DIE DEVICE CHECK
; L135
LOAD      M14580	// R_P&P CYCLE RUN
AND       P0005D	// R_P&P UP (SENSOR)
AND       P00160	// R_P&P 1st EJECT ON
AND       M01430	// R_IN BUF VC KP
AND NOT   M06616	// R_P&P 1st DET VAC ON
AND NOT   M1902F	// DRY RUN
OUT       M1461A	// R_1st PP VC ALARM
; L136
LOAD      M14580	// R_P&P CYCLE RUN
AND       P0005D	// R_P&P UP (SENSOR)
AND       P00162	// R_P&P 2nd EJECT ON
AND       M01431	// R_1st DIE VC KP
AND NOT   M06617	// R_P&P 2nd DET VAC ON
AND NOT   M1902F	// DRY RUN
OUT       M1461B	// R_2nd PP VC ALARM
; L137
LOAD      M14580	// R_P&P CYCLE RUN
AND       P0005D	// R_P&P UP (SENSOR)
AND       P00164	// R_P&P 3rd EJECT ON
AND       M01432	// R_2nd DIE VC KP
AND NOT   M06618	// R_P&P 3rd DET VAC ON
AND NOT   M1902F	// DRY RUN
OUT       M1461C	// R_3rd PP VC ALARM
; L138
LOAD      M14580	// R_P&P CYCLE RUN
AND       P0005D	// R_P&P UP (SENSOR)
AND       P00166	// R_P&P 4th EJECT ON
AND       M01433	// R_3rd DIE VC KP
AND NOT   M06619	// R_P&P 4th DET VAC ON
AND NOT   M1902F	// DRY RUN
OUT       M1461D	// R_4th PP VC ALARM
; L139
LOAD      M14580	// R_P&P CYCLE RUN
AND       P0005D	// R_P&P UP (SENSOR)
AND       P00168	// R_P&P 5th EJECT ON
AND       M01434	// R_4th DIE VC KP
AND NOT   M0661A	// R_P&P 5th DET VAC ON
AND NOT   M1902F	// DRY RUN
OUT       M1461E	// R_5th PP VC ALARM
// ========== 1st VACUUM ON/OFF ==========
; L141
LOAD      M14580	// R_P&P CYCLE RUN
AND       M14513	// R_P&P STEP#03
OR        M14812	// T)PP 1st VC ON
OR        M14620	// R_1st PP VC ON
AND NOT   M1451A	// R_P&P STEP#10
AND NOT   M14814	// T)PP 1st VC OFF
OUT       M14620	// R_1st PP VC ON

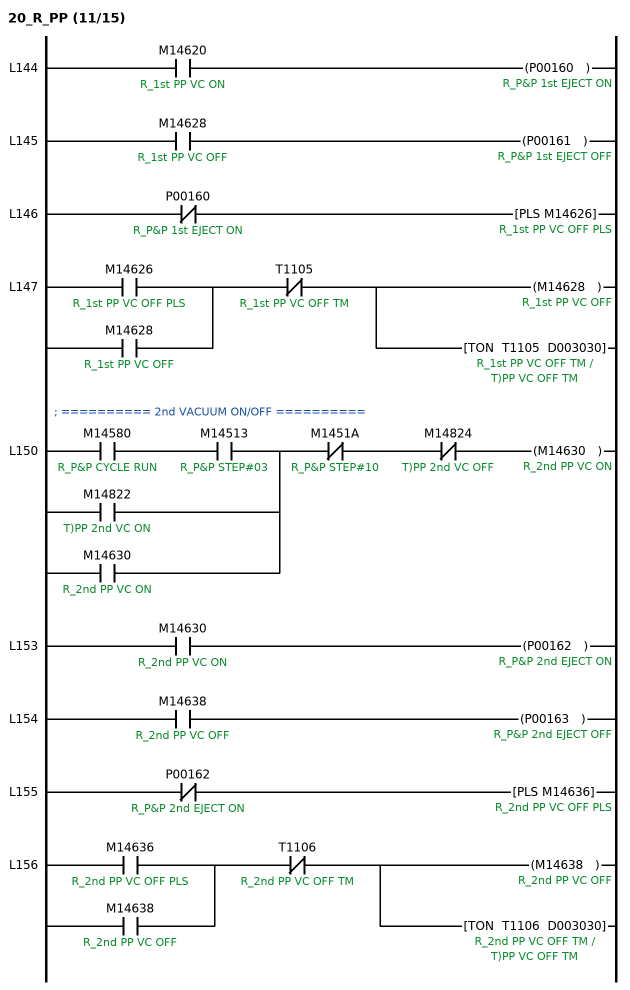
; L144
LOAD      M14620	// R_1st PP VC ON
OUT       P00160	// R_P&P 1st EJECT ON
; L145
LOAD      M14628	// R_1st PP VC OFF
OUT       P00161	// R_P&P 1st EJECT OFF
; L146
LOAD NOT  P00160	// R_P&P 1st EJECT ON
OUTP      M14626	// R_1st PP VC OFF PLS
; L147
LOAD      M14626	// R_1st PP VC OFF PLS
OR        M14628	// R_1st PP VC OFF
AND NOT   T1105	// R_1st PP VC OFF TM
OUT       M14628	// R_1st PP VC OFF
TON       T1105 D003030	// R_1st PP VC OFF TM / T)PP VC OFF TM
// ========== 2nd VACUUM ON/OFF ==========
; L150
LOAD      M14580	// R_P&P CYCLE RUN
AND       M14513	// R_P&P STEP#03
OR        M14822	// T)PP 2nd VC ON
OR        M14630	// R_2nd PP VC ON
AND NOT   M1451A	// R_P&P STEP#10
AND NOT   M14824	// T)PP 2nd VC OFF
OUT       M14630	// R_2nd PP VC ON
; L153
LOAD      M14630	// R_2nd PP VC ON
OUT       P00162	// R_P&P 2nd EJECT ON
; L154
LOAD      M14638	// R_2nd PP VC OFF
OUT       P00163	// R_P&P 2nd EJECT OFF
; L155
LOAD NOT  P00162	// R_P&P 2nd EJECT ON
OUTP      M14636	// R_2nd PP VC OFF PLS
; L156
LOAD      M14636	// R_2nd PP VC OFF PLS
OR        M14638	// R_2nd PP VC OFF
AND NOT   T1106	// R_2nd PP VC OFF TM
OUT       M14638	// R_2nd PP VC OFF
TON       T1106 D003030	// R_2nd PP VC OFF TM / T)PP VC OFF TM

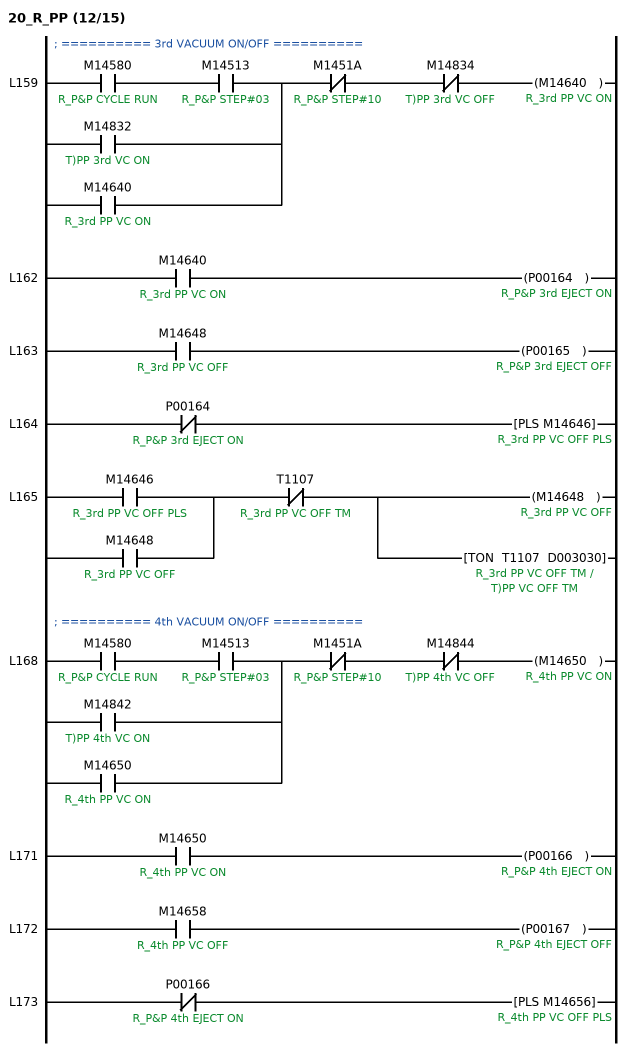
// ========== 3rd VACUUM ON/OFF ==========
; L159
LOAD      M14580	// R_P&P CYCLE RUN
AND       M14513	// R_P&P STEP#03
OR        M14832	// T)PP 3rd VC ON
OR        M14640	// R_3rd PP VC ON
AND NOT   M1451A	// R_P&P STEP#10
AND NOT   M14834	// T)PP 3rd VC OFF
OUT       M14640	// R_3rd PP VC ON
; L162
LOAD      M14640	// R_3rd PP VC ON
OUT       P00164	// R_P&P 3rd EJECT ON
; L163
LOAD      M14648	// R_3rd PP VC OFF
OUT       P00165	// R_P&P 3rd EJECT OFF
; L164
LOAD NOT  P00164	// R_P&P 3rd EJECT ON
OUTP      M14646	// R_3rd PP VC OFF PLS
; L165
LOAD      M14646	// R_3rd PP VC OFF PLS
OR        M14648	// R_3rd PP VC OFF
AND NOT   T1107	// R_3rd PP VC OFF TM
OUT       M14648	// R_3rd PP VC OFF
TON       T1107 D003030	// R_3rd PP VC OFF TM / T)PP VC OFF TM
// ========== 4th VACUUM ON/OFF ==========
; L168
LOAD      M14580	// R_P&P CYCLE RUN
AND       M14513	// R_P&P STEP#03
OR        M14842	// T)PP 4th VC ON
OR        M14650	// R_4th PP VC ON
AND NOT   M1451A	// R_P&P STEP#10
AND NOT   M14844	// T)PP 4th VC OFF
OUT       M14650	// R_4th PP VC ON
; L171
LOAD      M14650	// R_4th PP VC ON
OUT       P00166	// R_P&P 4th EJECT ON
; L172
LOAD      M14658	// R_4th PP VC OFF
OUT       P00167	// R_P&P 4th EJECT OFF
; L173
LOAD NOT  P00166	// R_P&P 4th EJECT ON
OUTP      M14656	// R_4th PP VC OFF PLS

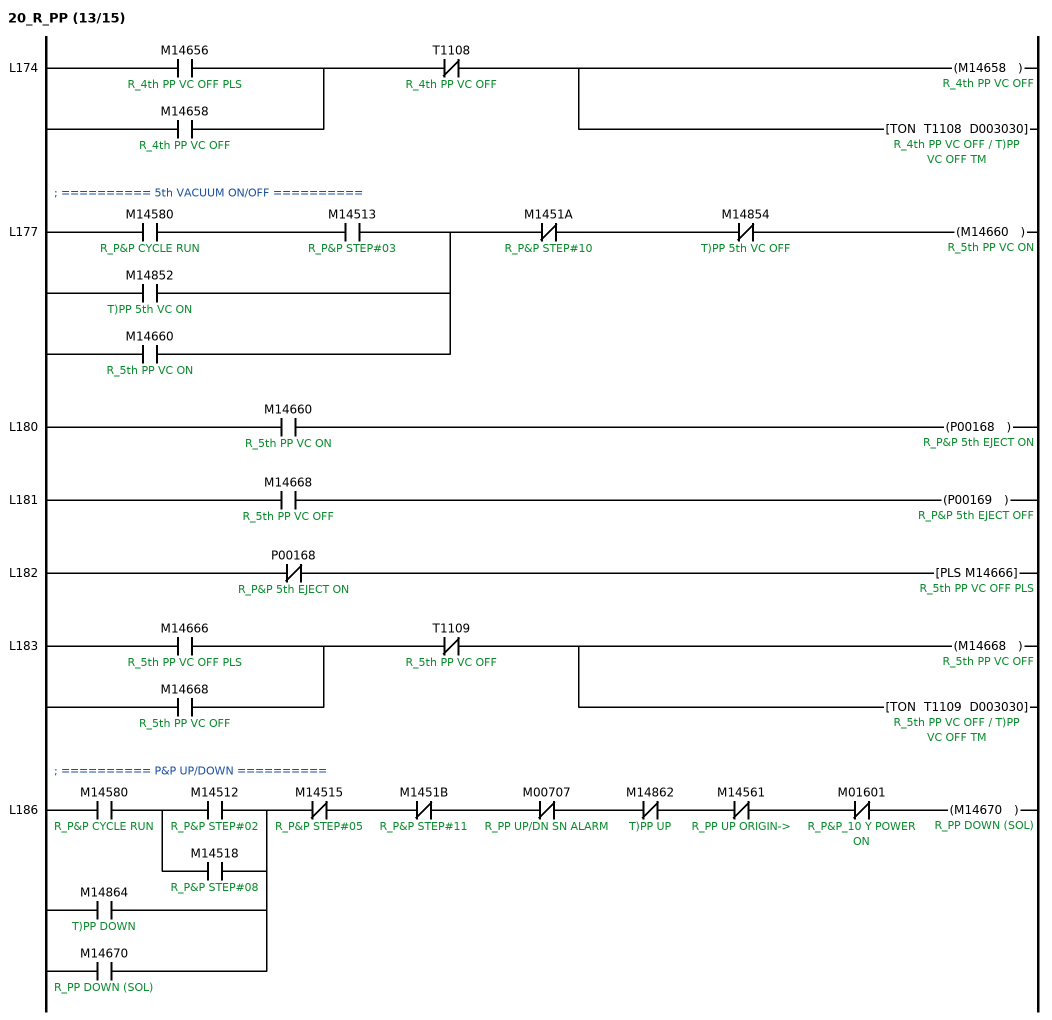
; L174
LOAD      M14656	// R_4th PP VC OFF PLS
OR        M14658	// R_4th PP VC OFF
AND NOT   T1108	// R_4th PP VC OFF
OUT       M14658	// R_4th PP VC OFF
TON       T1108 D003030	// R_4th PP VC OFF / T)PP VC OFF TM
// ========== 5th VACUUM ON/OFF ==========
; L177
LOAD      M14580	// R_P&P CYCLE RUN
AND       M14513	// R_P&P STEP#03
OR        M14852	// T)PP 5th VC ON
OR        M14660	// R_5th PP VC ON
AND NOT   M1451A	// R_P&P STEP#10
AND NOT   M14854	// T)PP 5th VC OFF
OUT       M14660	// R_5th PP VC ON
; L180
LOAD      M14660	// R_5th PP VC ON
OUT       P00168	// R_P&P 5th EJECT ON
; L181
LOAD      M14668	// R_5th PP VC OFF
OUT       P00169	// R_P&P 5th EJECT OFF
; L182
LOAD NOT  P00168	// R_P&P 5th EJECT ON
OUTP      M14666	// R_5th PP VC OFF PLS
; L183
LOAD      M14666	// R_5th PP VC OFF PLS
OR        M14668	// R_5th PP VC OFF
AND NOT   T1109	// R_5th PP VC OFF
OUT       M14668	// R_5th PP VC OFF
TON       T1109 D003030	// R_5th PP VC OFF / T)PP VC OFF TM
// ========== P&P UP/DOWN ==========
; L186
LOAD      M14580	// R_P&P CYCLE RUN
LOAD      M14512	// R_P&P STEP#02
OR        M14518	// R_P&P STEP#08
AND LOAD
OR        M14864	// T)PP DOWN
OR        M14670	// R_PP DOWN (SOL)
AND NOT   M14515	// R_P&P STEP#05
AND NOT   M1451B	// R_P&P STEP#11
AND NOT   M00707	// R_PP UP/DN SN ALARM
AND NOT   M14862	// T)PP UP
AND NOT   M14561	// R_PP UP ORIGIN->
AND NOT   M01601	// R_P&P_10 Y POWER ON
OUT       M14670	// R_PP DOWN (SOL)

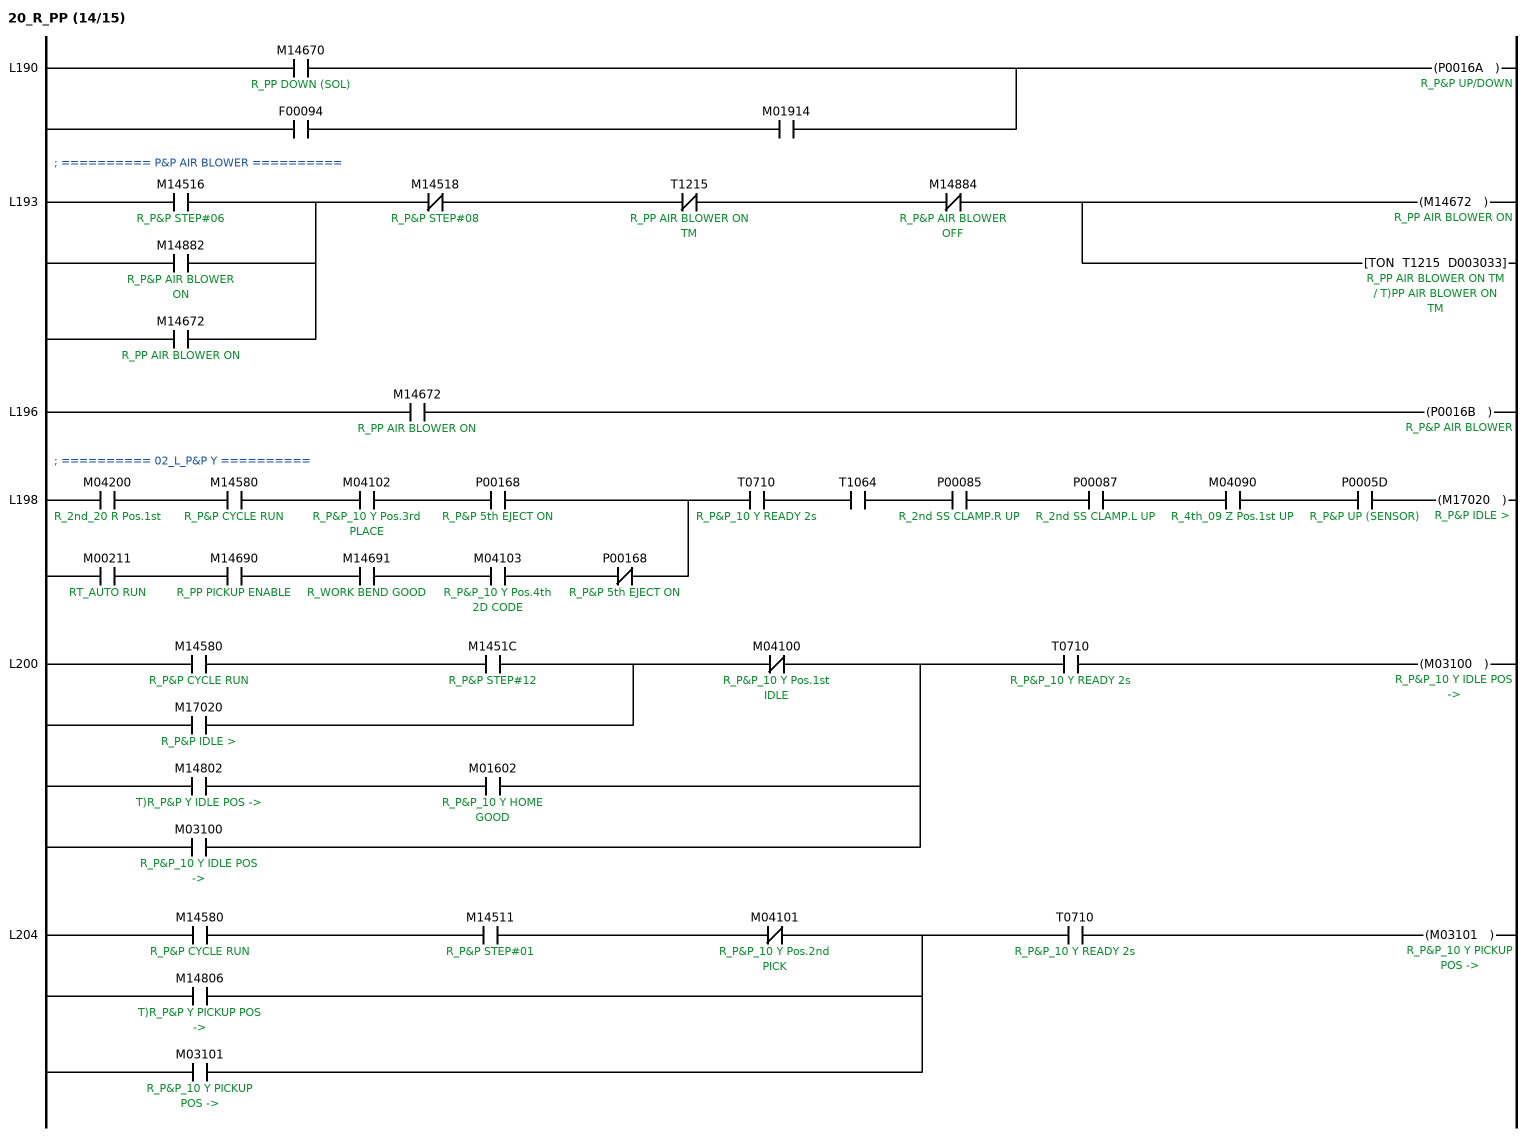
; L190
LOAD      M14670	// R_PP DOWN (SOL)
LOAD      F00094
AND       M01914
OR LOAD
OUT       P0016A	// R_P&P UP/DOWN
// ========== P&P AIR BLOWER ==========
; L193
LOAD      M14516	// R_P&P STEP#06
OR        M14882	// R_P&P AIR BLOWER ON
OR        M14672	// R_PP AIR BLOWER ON
AND NOT   M14518	// R_P&P STEP#08
AND NOT   T1215	// R_PP AIR BLOWER ON TM
AND NOT   M14884	// R_P&P AIR BLOWER OFF
OUT       M14672	// R_PP AIR BLOWER ON
TON       T1215 D003033	// R_PP AIR BLOWER ON TM / T)PP AIR BLOWER ON TM
; L196
LOAD      M14672	// R_PP AIR BLOWER ON
OUT       P0016B	// R_P&P AIR BLOWER
// ========== 02_L_P&P Y ==========
; L198
LOAD      M04200	// R_2nd_20 R Pos.1st
AND       M14580	// R_P&P CYCLE RUN
AND       M04102	// R_P&P_10 Y Pos.3rd PLACE
AND       P00168	// R_P&P 5th EJECT ON
LOAD      M00211	// RT_AUTO RUN
AND       M14690	// R_PP PICKUP ENABLE
AND       M14691	// R_WORK BEND GOOD
AND       M04103	// R_P&P_10 Y Pos.4th 2D CODE
AND NOT   P00168	// R_P&P 5th EJECT ON
OR LOAD
AND       T0710	// R_P&P_10 Y READY 2s
AND       T1064
AND       P00085	// R_2nd SS CLAMP.R UP
AND       P00087	// R_2nd SS CLAMP.L UP
AND       M04090	// R_4th_09 Z Pos.1st UP
AND       P0005D	// R_P&P UP (SENSOR)
OUT       M17020	// R_P&P IDLE >
; L200
LOAD      M14580	// R_P&P CYCLE RUN
AND       M1451C	// R_P&P STEP#12
OR        M17020	// R_P&P IDLE >
AND NOT   M04100	// R_P&P_10 Y Pos.1st IDLE
LOAD      M14802	// T)R_P&P Y IDLE POS ->
AND       M01602	// R_P&P_10 Y HOME GOOD
OR LOAD
OR        M03100	// R_P&P_10 Y IDLE POS ->
AND       T0710	// R_P&P_10 Y READY 2s
OUT       M03100	// R_P&P_10 Y IDLE POS ->
; L204
LOAD      M14580	// R_P&P CYCLE RUN
AND       M14511	// R_P&P STEP#01
AND NOT   M04101	// R_P&P_10 Y Pos.2nd PICK
OR        M14806	// T)R_P&P Y PICKUP POS ->
OR        M03101	// R_P&P_10 Y PICKUP POS ->
AND       T0710	// R_P&P_10 Y READY 2s
OUT       M03101	// R_P&P_10 Y PICKUP POS ->

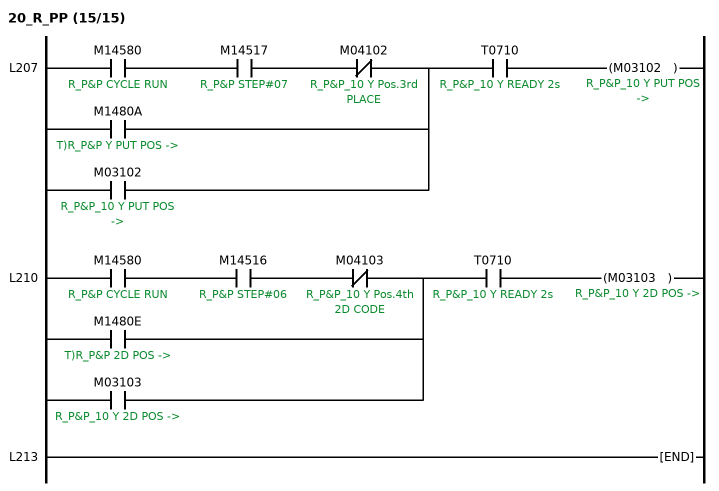
; L207
LOAD      M14580	// R_P&P CYCLE RUN
AND       M14517	// R_P&P STEP#07
AND NOT   M04102	// R_P&P_10 Y Pos.3rd PLACE
OR        M1480A	// T)R_P&P Y PUT POS ->
OR        M03102	// R_P&P_10 Y PUT POS ->
AND       T0710	// R_P&P_10 Y READY 2s
OUT       M03102	// R_P&P_10 Y PUT POS ->
; L210
LOAD      M14580	// R_P&P CYCLE RUN
AND       M14516	// R_P&P STEP#06
AND NOT   M04103	// R_P&P_10 Y Pos.4th 2D CODE
OR        M1480E	// T)R_P&P 2D POS ->
OR        M03103	// R_P&P_10 Y 2D POS ->
AND       T0710	// R_P&P_10 Y READY 2s
OUT       M03103	// R_P&P_10 Y 2D POS ->
; L213
END

PROGRAM 30_IN_LR_BUFFER (task: ½ºÄµ ÇÁ·Î±×·¥)

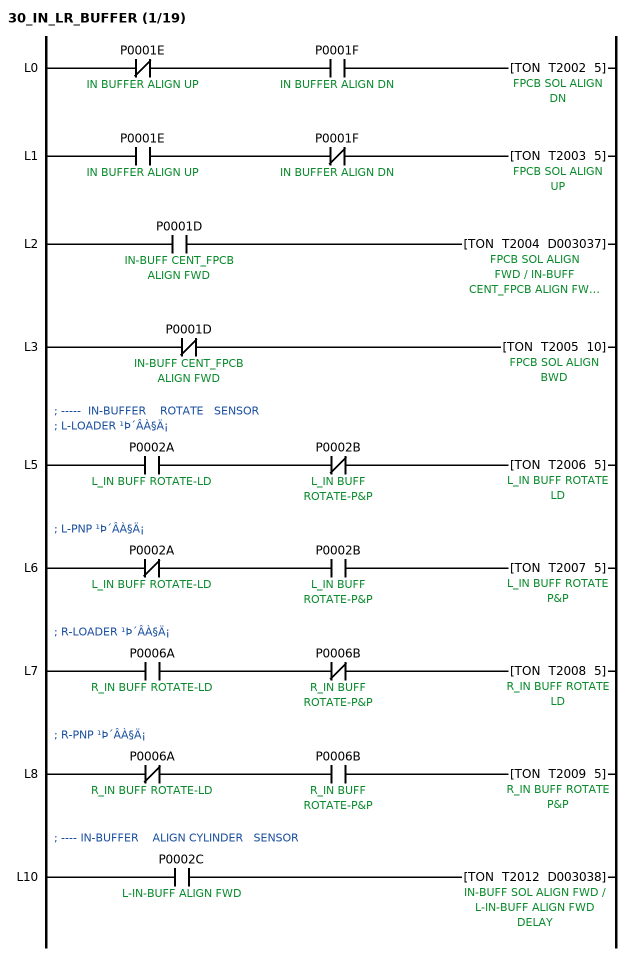
; L0
LOAD NOT  P0001E	// IN BUFFER ALIGN UP
AND       P0001F	// IN BUFFER ALIGN DN
TON       T2002 5	// FPCB SOL ALIGN        DN
; L1
LOAD      P0001E	// IN BUFFER ALIGN UP
AND NOT   P0001F	// IN BUFFER ALIGN DN
TON       T2003 5	// FPCB SOL ALIGN         UP
; L2
LOAD      P0001D	// IN-BUFF CENT_FPCB ALIGN FWD
TON       T2004 D003037	// FPCB SOL ALIGN         FWD / IN-BUFF CENT_FPCB ALIGN FWD DELAY
; L3
LOAD NOT  P0001D	// IN-BUFF CENT_FPCB ALIGN FWD
TON       T2005 10	// FPCB SOL ALIGN         BWD
// -----  IN-BUFFER    ROTATE   SENSOR
; L5
LOAD      P0002A	// L_IN BUFF ROTATE-LD
AND NOT   P0002B	// L_IN BUFF ROTATE-P&P
TON       T2006 5	// L_IN BUFF ROTATE     LD
// output comment: L-LOADER ¹Þ´ÂÀ§Ä¡
; L6
LOAD NOT  P0002A	// L_IN BUFF ROTATE-LD
AND       P0002B	// L_IN BUFF ROTATE-P&P
TON       T2007 5	// L_IN BUFF ROTATE      P&P
// output comment: L-PNP ¹Þ´ÂÀ§Ä¡
; L7
LOAD      P0006A	// R_IN BUFF ROTATE-LD
AND NOT   P0006B	// R_IN BUFF ROTATE-P&P
TON       T2008 5	// R_IN BUFF ROTATE      LD
// output comment: R-LOADER ¹Þ´ÂÀ§Ä¡
; L8
LOAD NOT  P0006A	// R_IN BUFF ROTATE-LD
AND       P0006B	// R_IN BUFF ROTATE-P&P
TON       T2009 5	// R_IN BUFF ROTATE      P&P
// output comment: R-PNP ¹Þ´ÂÀ§Ä¡
// ---- IN-BUFFER    ALIGN CYLINDER   SENSOR
; L10
LOAD      P0002C	// L-IN-BUFF ALIGN FWD
TON       T2012 D003038	// IN-BUFF SOL ALIGN FWD / L-IN-BUFF ALIGN FWD DELAY

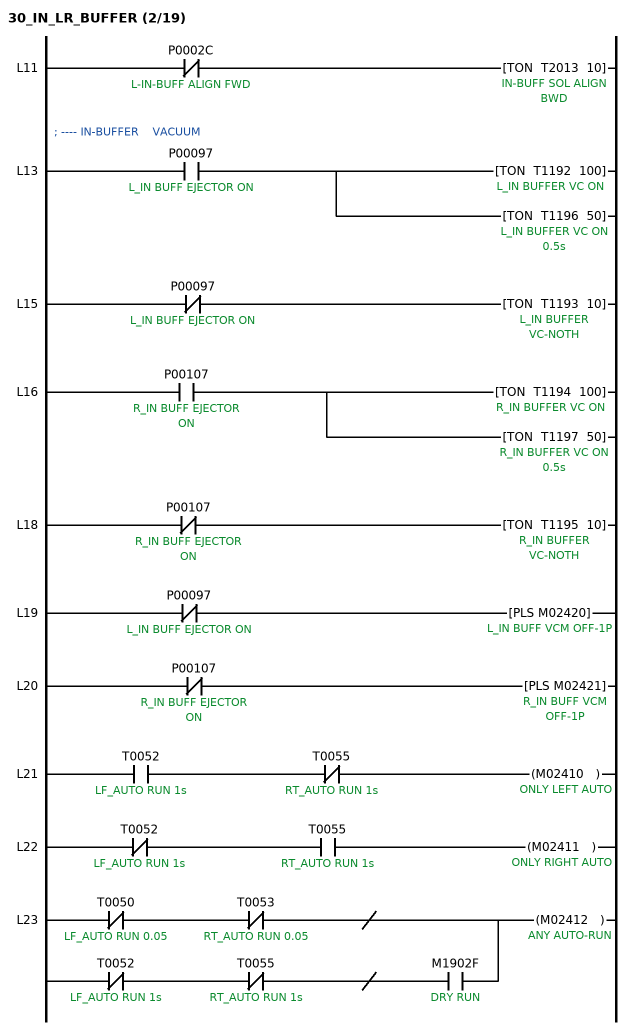
; L11
LOAD NOT  P0002C	// L-IN-BUFF ALIGN FWD
TON       T2013 10	// IN-BUFF SOL ALIGN BWD
// ---- IN-BUFFER    VACUUM
; L13
LOAD      P00097	// L_IN BUFF EJECTOR ON
TON       T1192 100	// L_IN BUFFER VC ON
TON       T1196 50	// L_IN BUFFER VC ON 0.5s
; L15
LOAD NOT  P00097	// L_IN BUFF EJECTOR ON
TON       T1193 10	// L_IN BUFFER VC-NOTH
; L16
LOAD      P00107	// R_IN BUFF EJECTOR ON
TON       T1194 100	// R_IN BUFFER VC ON
TON       T1197 50	// R_IN BUFFER VC ON 0.5s
; L18
LOAD NOT  P00107	// R_IN BUFF EJECTOR ON
TON       T1195 10	// R_IN BUFFER VC-NOTH
; L19
LOAD NOT  P00097	// L_IN BUFF EJECTOR ON
OUTP      M02420	// L_IN BUFF VCM OFF-1P
; L20
LOAD NOT  P00107	// R_IN BUFF EJECTOR ON
OUTP      M02421	// R_IN BUFF VCM OFF-1P
; L21
LOAD      T0052	// LF_AUTO RUN 1s
AND NOT   T0055	// RT_AUTO RUN 1s
OUT       M02410	// ONLY LEFT AUTO
; L22
LOAD NOT  T0052	// LF_AUTO RUN 1s
AND       T0055	// RT_AUTO RUN 1s
OUT       M02411	// ONLY RIGHT AUTO
; L23
LOAD NOT  T0050	// LF_AUTO RUN 0.05
AND NOT   T0053	// RT_AUTO RUN 0.05
NOT
LOAD NOT  T0052	// LF_AUTO RUN 1s
AND NOT   T0055	// RT_AUTO RUN 1s
NOT
AND       M1902F	// DRY RUN
OR LOAD
OUT       M02412	// ANY AUTO-RUN

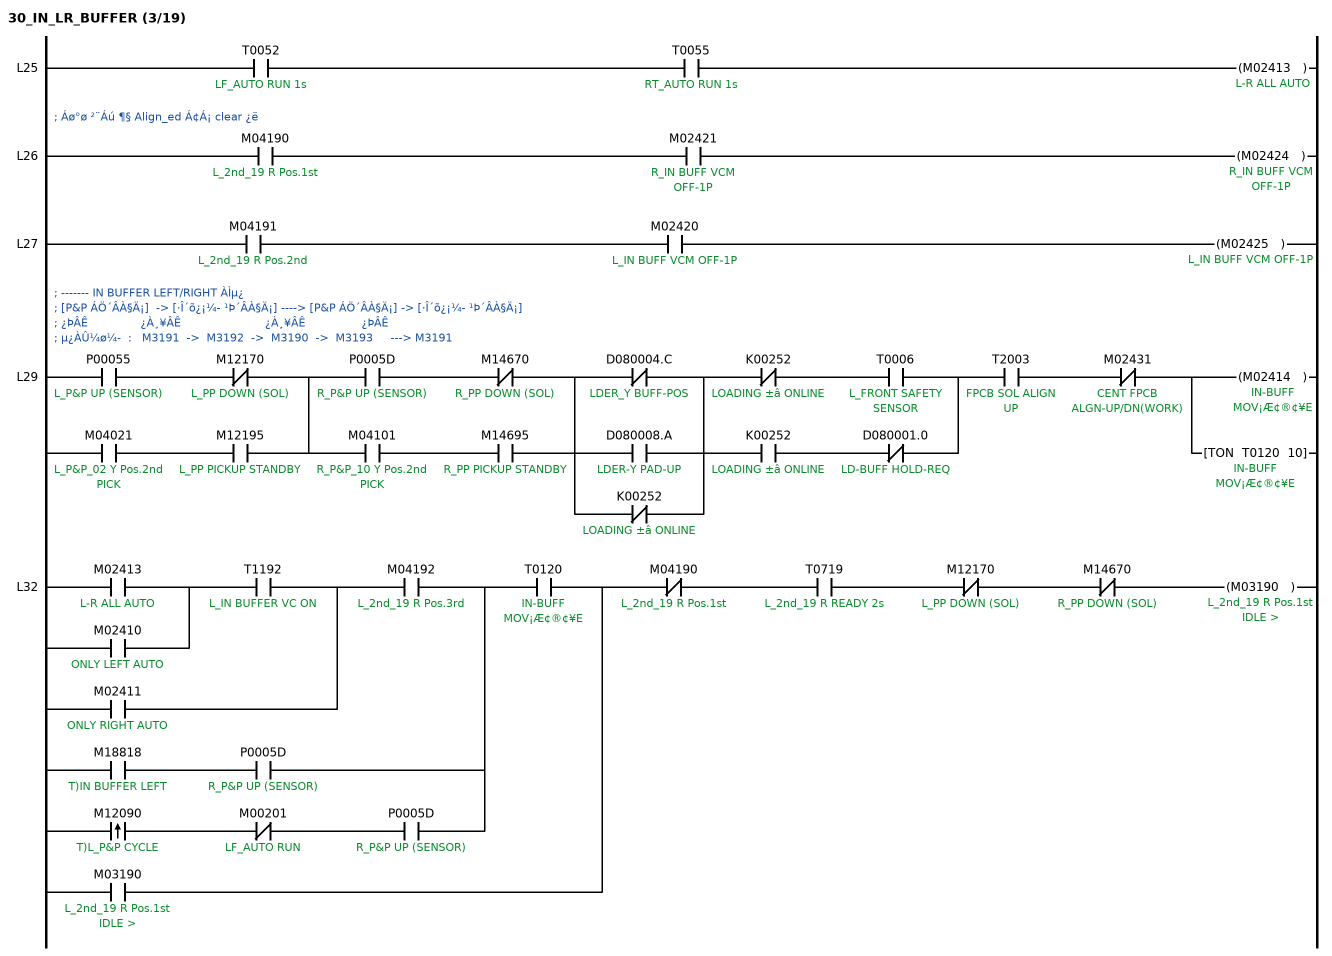
; L25
LOAD      T0052	// LF_AUTO RUN 1s
AND       T0055	// RT_AUTO RUN 1s
OUT       M02413	// L-R ALL AUTO
; L26
LOAD      M04190	// L_2nd_19 R Pos.1st 
AND       M02421	// R_IN BUFF VCM OFF-1P
OUT       M02424	// R_IN BUFF VCM OFF-1P
// output comment: Áø°ø ²¨Áú ¶§ Align_ed Á¢Á¡ clear ¿ë
; L27
LOAD      M04191	// L_2nd_19 R Pos.2nd
AND       M02420	// L_IN BUFF VCM OFF-1P
OUT       M02425	// L_IN BUFF VCM OFF-1P
// ------- IN BUFFER LEFT/RIGHT ÀÌµ¿
// 
// 
//  [P&P ÁÖ´ÂÀ§Ä¡]  -> [·Î´õ¿¡¼­ ¹Þ´ÂÀ§Ä¡] ----> [P&P ÁÖ´ÂÀ§Ä¡] -> [·Î´õ¿¡¼­ ¹Þ´ÂÀ§Ä¡]
//   ¿ÞÂÊ               ¿À¸¥ÂÊ                        ¿À¸¥ÂÊ                ¿ÞÂÊ
//     
//  µ¿ÀÛ¼ø¼­  :   M3191  ->  M3192  ->  M3190  ->  M3193     ---> M3191
; L29
LOAD      P00055	// L_P&P UP (SENSOR)
AND NOT   M12170	// L_PP DOWN (SOL)
LOAD      M04021	// L_P&P_02 Y Pos.2nd PICK
AND       M12195	// L_PP PICKUP STANDBY
OR LOAD
LOAD      P0005D	// R_P&P UP (SENSOR)
AND NOT   M14670	// R_PP DOWN (SOL)
LOAD      M04101	// R_P&P_10 Y Pos.2nd PICK
AND       M14695	// R_PP PICKUP STANDBY
OR LOAD
AND LOAD
LOAD NOT  D080004.C	// LDER_Y BUFF-POS
OR        D080008.A	// LDER-Y PAD-UP
OR NOT    K00252	// LOADING ±â ONLINE
AND LOAD
LOAD NOT  K00252	// LOADING ±â ONLINE
AND       T0006	// L_FRONT SAFETY SENSOR
LOAD      K00252	// LOADING ±â ONLINE
AND NOT   D080001.0	// LD-BUFF HOLD-REQ
OR LOAD
AND LOAD
AND       T2003	// FPCB SOL ALIGN         UP
AND NOT   M02431	// CENT FPCB ALGN-UP/DN(WORK)
OUT       M02414	// IN-BUFF MOV¡Æ¢®¢¥E
TON       T0120 10	// IN-BUFF MOV¡Æ¢®¢¥E
; L32
LOAD      M02413	// L-R ALL AUTO
OR        M02410	// ONLY LEFT AUTO
AND       T1192	// L_IN BUFFER VC ON
OR        M02411	// ONLY RIGHT AUTO
AND       M04192	// L_2nd_19 R Pos.3rd
LOAD      M18818	// T)IN BUFFER LEFT
AND       P0005D	// R_P&P UP (SENSOR)
OR LOAD
LOADP     M12090	// T)L_P&P CYCLE
AND NOT   M00201	// LF_AUTO RUN
AND       P0005D	// R_P&P UP (SENSOR)
OR LOAD
AND       T0120	// IN-BUFF MOV¡Æ¢®¢¥E
OR        M03190	// L_2nd_19 R Pos.1st IDLE >
AND NOT   M04190	// L_2nd_19 R Pos.1st 
AND       T0719	// L_2nd_19 R READY 2s
AND NOT   M12170	// L_PP DOWN (SOL)
AND NOT   M14670	// R_PP DOWN (SOL)
OUT       M03190	// L_2nd_19 R Pos.1st IDLE >

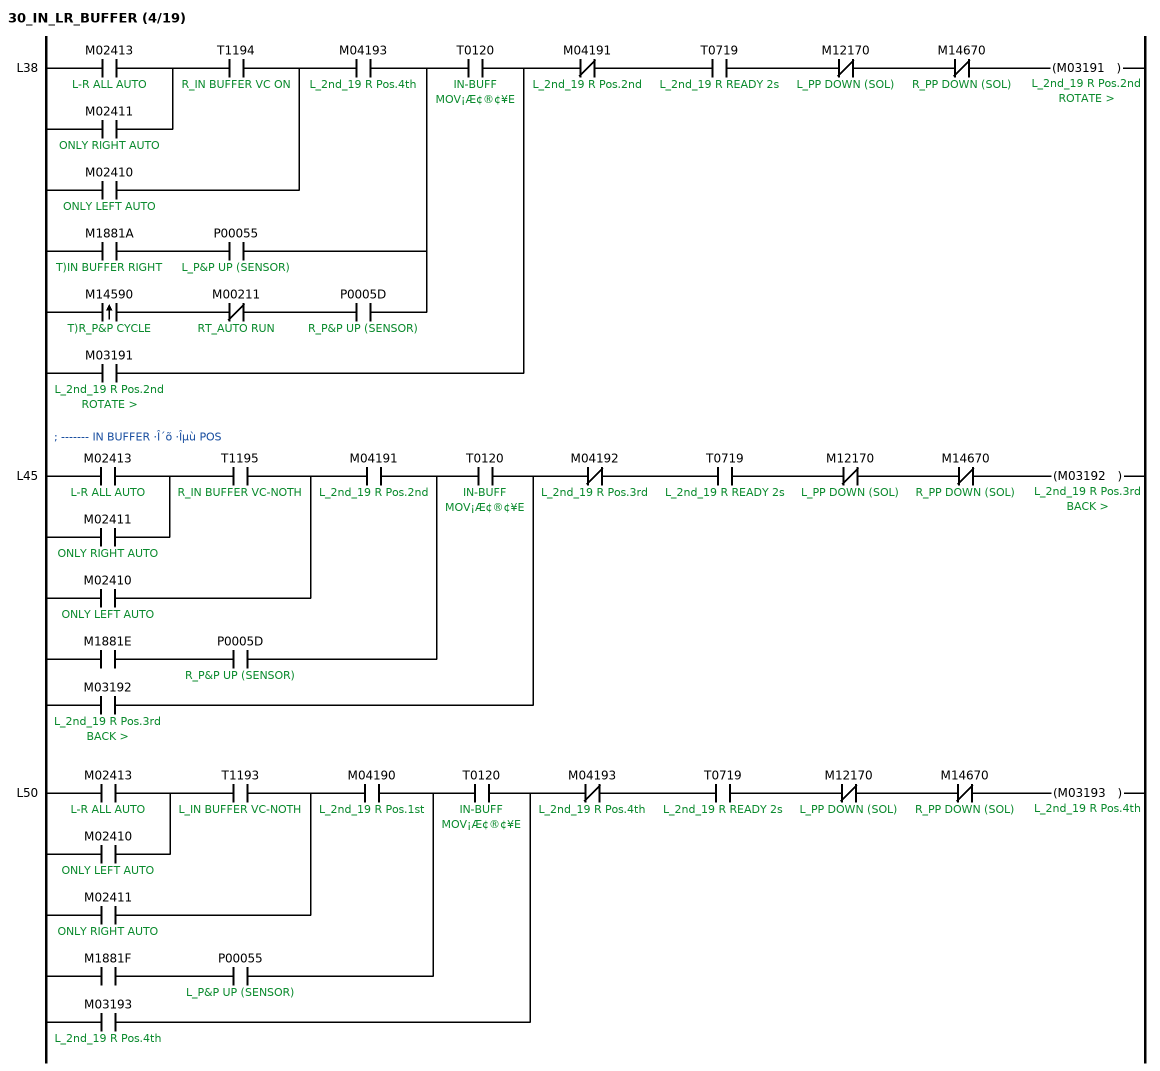
; L38
LOAD      M02413	// L-R ALL AUTO
OR        M02411	// ONLY RIGHT AUTO
AND       T1194	// R_IN BUFFER VC ON
OR        M02410	// ONLY LEFT AUTO
AND       M04193	// L_2nd_19 R Pos.4th 
LOAD      M1881A	// T)IN BUFFER RIGHT
AND       P00055	// L_P&P UP (SENSOR)
OR LOAD
LOADP     M14590	// T)R_P&P CYCLE
AND NOT   M00211	// RT_AUTO RUN
AND       P0005D	// R_P&P UP (SENSOR)
OR LOAD
AND       T0120	// IN-BUFF MOV¡Æ¢®¢¥E
OR        M03191	// L_2nd_19 R Pos.2nd ROTATE >
AND NOT   M04191	// L_2nd_19 R Pos.2nd
AND       T0719	// L_2nd_19 R READY 2s
AND NOT   M12170	// L_PP DOWN (SOL)
AND NOT   M14670	// R_PP DOWN (SOL)
OUT       M03191	// L_2nd_19 R Pos.2nd ROTATE >
// ------- IN BUFFER ·Î´õ ·Îµù POS
; L45
LOAD      M02413	// L-R ALL AUTO
OR        M02411	// ONLY RIGHT AUTO
AND       T1195	// R_IN BUFFER VC-NOTH
OR        M02410	// ONLY LEFT AUTO
AND       M04191	// L_2nd_19 R Pos.2nd
LOAD      M1881E
AND       P0005D	// R_P&P UP (SENSOR)
OR LOAD
AND       T0120	// IN-BUFF MOV¡Æ¢®¢¥E
OR        M03192	// L_2nd_19 R Pos.3rd BACK >
AND NOT   M04192	// L_2nd_19 R Pos.3rd
AND       T0719	// L_2nd_19 R READY 2s
AND NOT   M12170	// L_PP DOWN (SOL)
AND NOT   M14670	// R_PP DOWN (SOL)
OUT       M03192	// L_2nd_19 R Pos.3rd BACK >
; L50
LOAD      M02413	// L-R ALL AUTO
OR        M02410	// ONLY LEFT AUTO
AND       T1193	// L_IN BUFFER VC-NOTH
OR        M02411	// ONLY RIGHT AUTO
AND       M04190	// L_2nd_19 R Pos.1st 
LOAD      M1881F
AND       P00055	// L_P&P UP (SENSOR)
OR LOAD
AND       T0120	// IN-BUFF MOV¡Æ¢®¢¥E
OR        M03193	// L_2nd_19 R Pos.4th 
AND NOT   M04193	// L_2nd_19 R Pos.4th 
AND       T0719	// L_2nd_19 R READY 2s
AND NOT   M12170	// L_PP DOWN (SOL)
AND NOT   M14670	// R_PP DOWN (SOL)
OUT       M03193	// L_2nd_19 R Pos.4th 

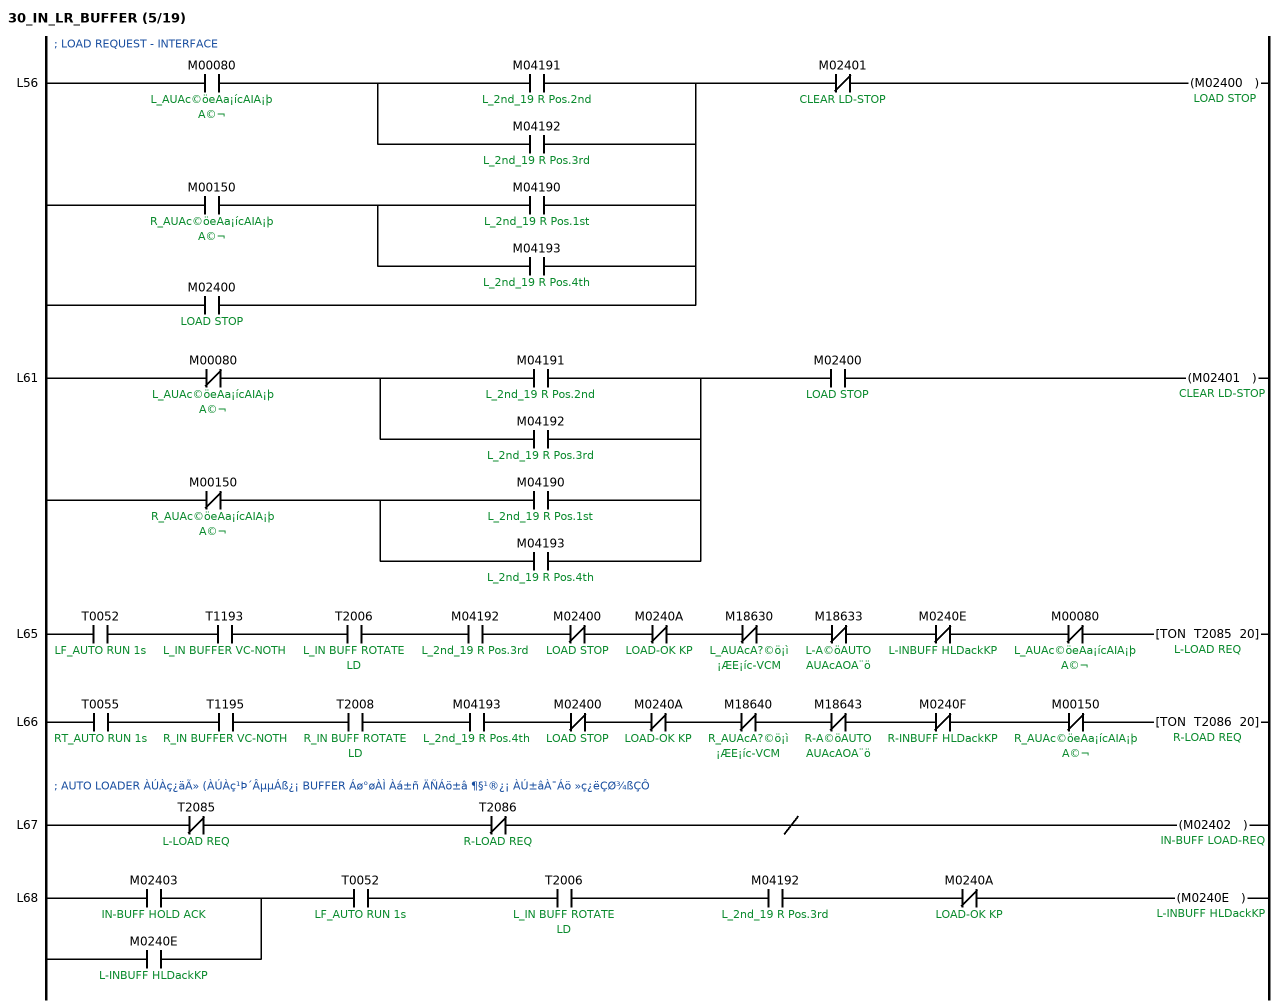
// LOAD REQUEST - INTERFACE
; L56
LOAD      M00080	// L_AUAc©öeAa¡ícAIA¡þA©¬
LOAD      M04191	// L_2nd_19 R Pos.2nd
OR        M04192	// L_2nd_19 R Pos.3rd
AND LOAD
LOAD      M00150	// R_AUAc©öeAa¡ícAIA¡þA©¬
LOAD      M04190	// L_2nd_19 R Pos.1st 
OR        M04193	// L_2nd_19 R Pos.4th 
AND LOAD
OR LOAD
OR        M02400	// LOAD STOP
AND NOT   M02401	// CLEAR LD-STOP
OUT       M02400	// LOAD STOP
; L61
LOAD NOT  M00080	// L_AUAc©öeAa¡ícAIA¡þA©¬
LOAD      M04191	// L_2nd_19 R Pos.2nd
OR        M04192	// L_2nd_19 R Pos.3rd
AND LOAD
LOAD NOT  M00150	// R_AUAc©öeAa¡ícAIA¡þA©¬
LOAD      M04190	// L_2nd_19 R Pos.1st 
OR        M04193	// L_2nd_19 R Pos.4th 
AND LOAD
OR LOAD
AND       M02400	// LOAD STOP
OUT       M02401	// CLEAR LD-STOP
; L65
LOAD      T0052	// LF_AUTO RUN 1s
AND       T1193	// L_IN BUFFER VC-NOTH
AND       T2006	// L_IN BUFF ROTATE     LD
AND       M04192	// L_2nd_19 R Pos.3rd
AND NOT   M02400	// LOAD STOP
AND NOT   M0240A	// LOAD-OK KP
AND NOT   M18630	// L_AUAcA?©ö¡ì ¡ÆE¡íc-VCM
AND NOT   M18633	// L-A©öAUTO AUAcAOA¨ö
AND NOT   M0240E	// L-INBUFF HLDackKP
AND NOT   M00080	// L_AUAc©öeAa¡ícAIA¡þA©¬
TON       T2085 20	// L-LOAD REQ
; L66
LOAD      T0055	// RT_AUTO RUN 1s
AND       T1195	// R_IN BUFFER VC-NOTH
AND       T2008	// R_IN BUFF ROTATE      LD
AND       M04193	// L_2nd_19 R Pos.4th 
AND NOT   M02400	// LOAD STOP
AND NOT   M0240A	// LOAD-OK KP
AND NOT   M18640	// R_AUAcA?©ö¡ì ¡ÆE¡íc-VCM
AND NOT   M18643	// R-A©öAUTO AUAcAOA¨ö
AND NOT   M0240F	// R-INBUFF HLDackKP
AND NOT   M00150	// R_AUAc©öeAa¡ícAIA¡þA©¬
TON       T2086 20	// R-LOAD REQ
; L67
LOAD NOT  T2085	// L-LOAD REQ
AND NOT   T2086	// R-LOAD REQ
NOT
OUT       M02402	// IN-BUFF LOAD-REQ
// output comment: AUTO LOADER ÀÚÀç¿äÃ» (ÀÚÀç¹Þ´ÂµµÁß¿¡ BUFFER Áø°øÀÌ Àá±ñ ÄÑÁö±â ¶§¹®¿¡ ÀÚ±âÀ¯Áö »ç¿ëÇØ¾ßÇÔ
; L68
LOAD      M02403	// IN-BUFF HOLD ACK
OR        M0240E	// L-INBUFF HLDackKP
AND       T0052	// LF_AUTO RUN 1s
AND       T2006	// L_IN BUFF ROTATE     LD
AND       M04192	// L_2nd_19 R Pos.3rd
AND NOT   M0240A	// LOAD-OK KP
OUT       M0240E	// L-INBUFF HLDackKP

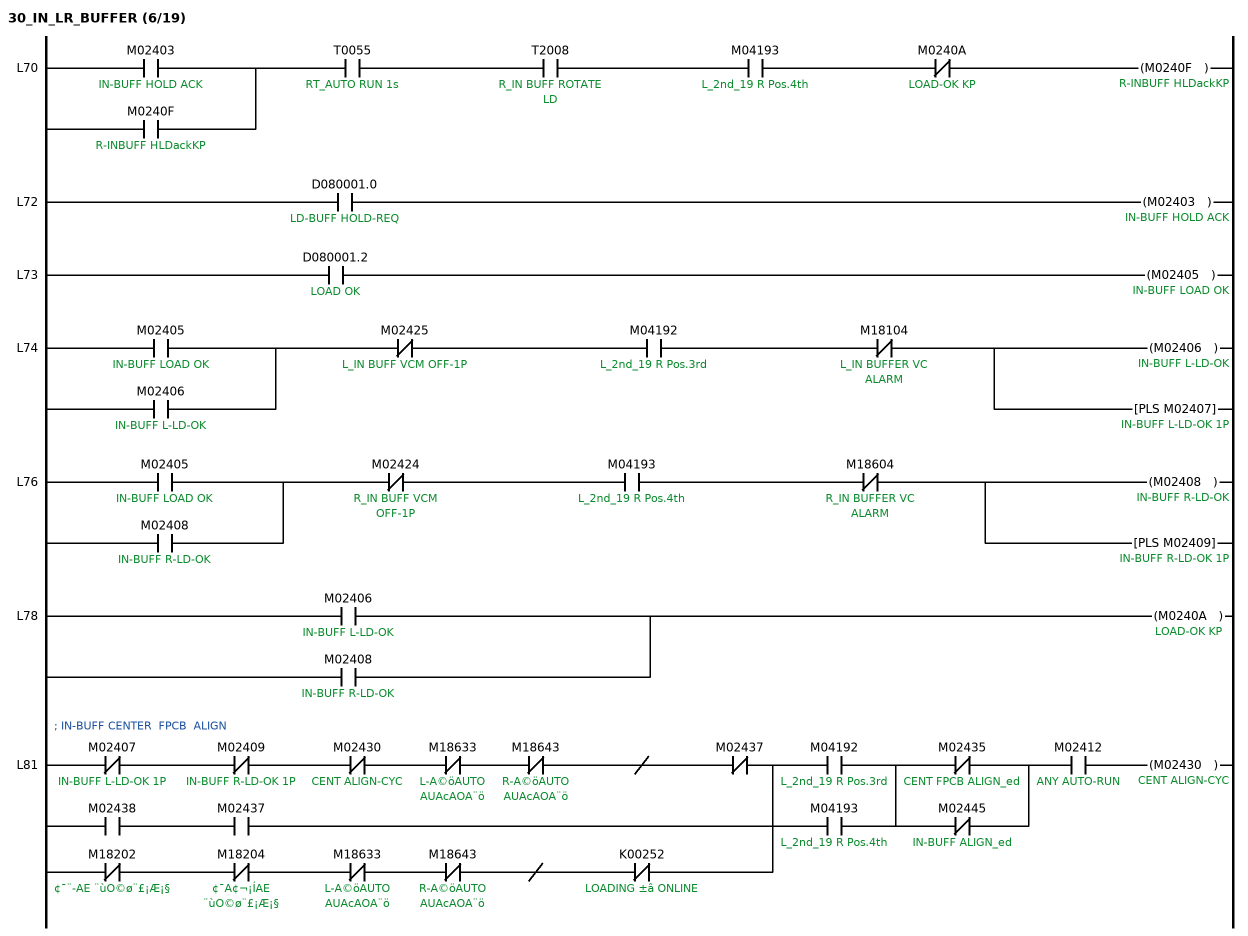
; L70
LOAD      M02403	// IN-BUFF HOLD ACK
OR        M0240F	// R-INBUFF HLDackKP
AND       T0055	// RT_AUTO RUN 1s
AND       T2008	// R_IN BUFF ROTATE      LD
AND       M04193	// L_2nd_19 R Pos.4th 
AND NOT   M0240A	// LOAD-OK KP
OUT       M0240F	// R-INBUFF HLDackKP
; L72
LOAD      D080001.0	// LD-BUFF HOLD-REQ
OUT       M02403	// IN-BUFF HOLD ACK
; L73
LOAD      D080001.2	// LOAD OK
OUT       M02405	// IN-BUFF LOAD OK
; L74
LOAD      M02405	// IN-BUFF LOAD OK
OR        M02406	// IN-BUFF L-LD-OK
AND NOT   M02425	// L_IN BUFF VCM OFF-1P
AND       M04192	// L_2nd_19 R Pos.3rd
AND NOT   M18104	// L_IN BUFFER VC ALARM
OUT       M02406	// IN-BUFF L-LD-OK
OUTP      M02407	// IN-BUFF L-LD-OK 1P
; L76
LOAD      M02405	// IN-BUFF LOAD OK
OR        M02408	// IN-BUFF R-LD-OK
AND NOT   M02424	// R_IN BUFF VCM OFF-1P
AND       M04193	// L_2nd_19 R Pos.4th 
AND NOT   M18604	// R_IN BUFFER VC ALARM
OUT       M02408	// IN-BUFF R-LD-OK
OUTP      M02409	// IN-BUFF R-LD-OK 1P
; L78
LOAD      M02406	// IN-BUFF L-LD-OK
OR        M02408	// IN-BUFF R-LD-OK
OUT       M0240A	// LOAD-OK KP
// IN-BUFF CENTER  FPCB  ALIGN
; L81
LOAD NOT  M02407	// IN-BUFF L-LD-OK 1P
AND NOT   M02409	// IN-BUFF R-LD-OK 1P
AND NOT   M02430	// CENT ALIGN-CYC
AND NOT   M18633	// L-A©öAUTO AUAcAOA¨ö
AND NOT   M18643	// R-A©öAUTO AUAcAOA¨ö
NOT
AND NOT   M02437
LOAD      M02438
AND       M02437
OR LOAD
LOAD NOT  M18202	// ¢¯¨­AE ¨ùO©ø¨£¡Æ¡§
AND NOT   M18204	// ¢¯A¢¬¡ÍAE ¨ùO©ø¨£¡Æ¡§
AND NOT   M18633	// L-A©öAUTO AUAcAOA¨ö
AND NOT   M18643	// R-A©öAUTO AUAcAOA¨ö
NOT
AND NOT   K00252	// LOADING ±â ONLINE
OR LOAD
LOAD      M04192	// L_2nd_19 R Pos.3rd
OR        M04193	// L_2nd_19 R Pos.4th 
AND LOAD
LOAD NOT  M02435	// CENT FPCB ALIGN_ed
OR NOT    M02445	// IN-BUFF ALIGN_ed
AND LOAD
AND       M02412	// ANY AUTO-RUN
OUT       M02430	// CENT ALIGN-CYC

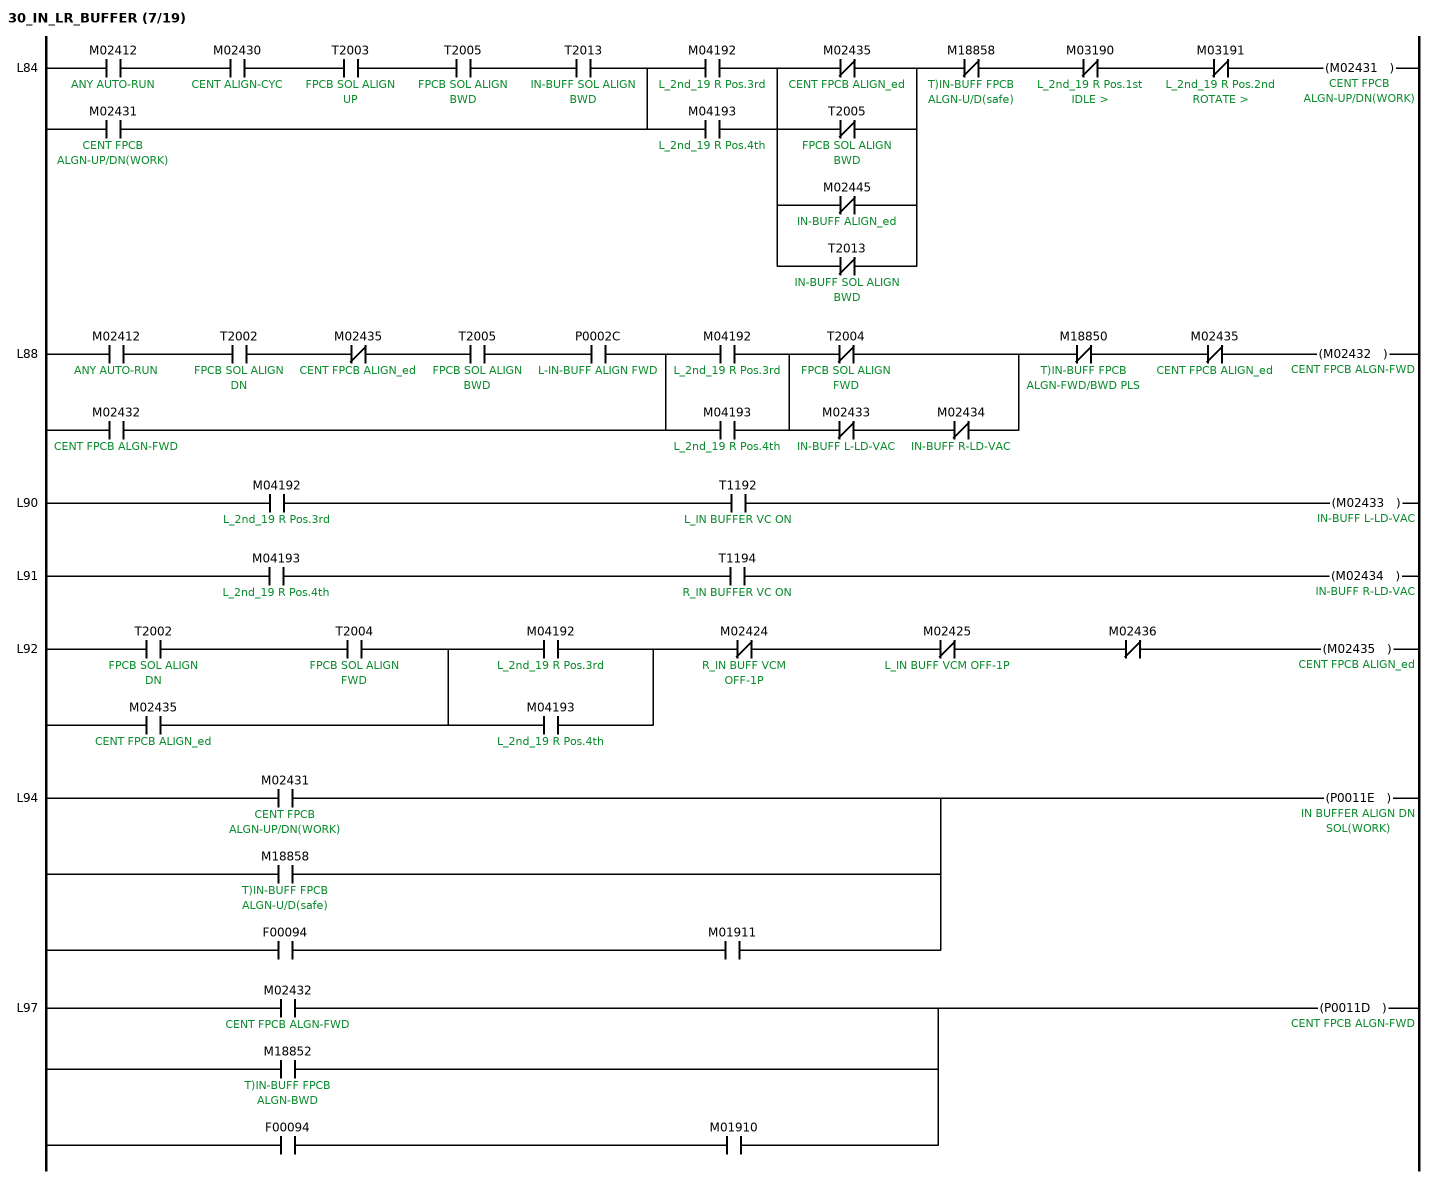
; L84
LOAD      M02412	// ANY AUTO-RUN
AND       M02430	// CENT ALIGN-CYC
AND       T2003	// FPCB SOL ALIGN         UP
AND       T2005	// FPCB SOL ALIGN         BWD
AND       T2013	// IN-BUFF SOL ALIGN BWD
OR        M02431	// CENT FPCB ALGN-UP/DN(WORK)
LOAD      M04192	// L_2nd_19 R Pos.3rd
OR        M04193	// L_2nd_19 R Pos.4th 
AND LOAD
LOAD NOT  M02435	// CENT FPCB ALIGN_ed
OR NOT    T2005	// FPCB SOL ALIGN         BWD
OR NOT    M02445	// IN-BUFF ALIGN_ed
OR NOT    T2013	// IN-BUFF SOL ALIGN BWD
AND LOAD
AND NOT   M18858	// T)IN-BUFF FPCB ALGN-U/D(safe)
AND NOT   M03190	// L_2nd_19 R Pos.1st IDLE >
AND NOT   M03191	// L_2nd_19 R Pos.2nd ROTATE >
OUT       M02431	// CENT FPCB ALGN-UP/DN(WORK)
; L88
LOAD      M02412	// ANY AUTO-RUN
AND       T2002	// FPCB SOL ALIGN        DN
AND NOT   M02435	// CENT FPCB ALIGN_ed
AND       T2005	// FPCB SOL ALIGN         BWD
AND       P0002C	// L-IN-BUFF ALIGN FWD
OR        M02432	// CENT FPCB ALGN-FWD
LOAD      M04192	// L_2nd_19 R Pos.3rd
OR        M04193	// L_2nd_19 R Pos.4th 
AND LOAD
LOAD NOT  T2004	// FPCB SOL ALIGN         FWD
LOAD NOT  M02433	// IN-BUFF L-LD-VAC
AND NOT   M02434	// IN-BUFF R-LD-VAC
OR LOAD
AND LOAD
AND NOT   M18850	// T)IN-BUFF FPCB ALGN-FWD/BWD PLS
AND NOT   M02435	// CENT FPCB ALIGN_ed
OUT       M02432	// CENT FPCB ALGN-FWD
; L90
LOAD      M04192	// L_2nd_19 R Pos.3rd
AND       T1192	// L_IN BUFFER VC ON
OUT       M02433	// IN-BUFF L-LD-VAC
; L91
LOAD      M04193	// L_2nd_19 R Pos.4th 
AND       T1194	// R_IN BUFFER VC ON
OUT       M02434	// IN-BUFF R-LD-VAC
; L92
LOAD      T2002	// FPCB SOL ALIGN        DN
AND       T2004	// FPCB SOL ALIGN         FWD
OR        M02435	// CENT FPCB ALIGN_ed
LOAD      M04192	// L_2nd_19 R Pos.3rd
OR        M04193	// L_2nd_19 R Pos.4th 
AND LOAD
AND NOT   M02424	// R_IN BUFF VCM OFF-1P
AND NOT   M02425	// L_IN BUFF VCM OFF-1P
AND NOT   M02436
OUT       M02435	// CENT FPCB ALIGN_ed
; L94
LOAD      M02431	// CENT FPCB ALGN-UP/DN(WORK)
OR        M18858	// T)IN-BUFF FPCB ALGN-U/D(safe)
LOAD      F00094
AND       M01911
OR LOAD
OUT       P0011E	// IN BUFFER ALIGN DN SOL(WORK)
; L97
LOAD      M02432	// CENT FPCB ALGN-FWD
OR        M18852	// T)IN-BUFF FPCB ALGN-BWD
LOAD      F00094
AND       M01910
OR LOAD
OUT       P0011D	// CENT FPCB ALGN-FWD

